LIN {X 0,Y 401.076,Z 526.774,A -85,B 0,C 180,E1 -11232.866,E2 -11232.866} C_VEL
LIN {X 0,Y 400.137,Z 539.303,A -85,B 0,C 180,E1 -11233.547,E2 -11233.547} C_VEL
LIN {X 0,Y 399.29,Z 551.619,A -85,B 0,C 180,E1 -11234.43,E2 -11234.43} C_VEL
LIN {X 0,Y 398.339,Z 562.751,A -85,B 0,C 180,E1 -11235.438,E2 -11235.438} C_VEL
LIN {X 0,Y 397.548,Z 573.979,A -85,B 0,C 180,E1 -11236.713,E2 -11236.713} C_VEL
LIN {X 0,Y 397.078,Z 581.427,A -85,B 0,C 180,E1 -11237.737,E2 -11237.737} C_VEL
LIN {X 0,Y 396.635,Z 590.764,A -85,B 0,C 180,E1 -11239.277,E2 -11239.277} C_VEL
LIN {X 0,Y 396.29,Z 600.831,A -85,B 0,C 180,E1 -11241.33,E2 -11241.33} C_VEL
LIN {X 0,Y 396.234,Z 606.786,A -85,B 0,C 180,E1 -11242.868,E2 -11242.868} C_VEL
LIN {X 0,Y 396.252,Z 611.402,A -85,B 0,C 180,E1 -11244.402,E2 -11244.402} C_VEL
LIN {X 0,Y 396.439,Z 614.849,A -85,B 0,C 180,E1 -11245.933,E2 -11245.933} C_VEL
LIN {X 0,Y 396.415,Z 616.498,A -85,B 0,C 180,E1 -11246.951,E2 -11246.951} C_VEL
LIN {X 0,Y 396.382,Z 617.7,A -85,B 0,C 180,E1 -11247.968,E2 -11247.968} C_VEL
LIN {X 0,Y 396.396,Z 618.449,A -85,B 0,C 180,E1 -11248.984,E2 -11248.984} C_VEL
LIN {X 0,Y 396.436,Z 618.72,A -85,B 0,C 180,E1 -11250,E2 -11250} C_VEL
LIN {X 0,Y 396.383,Z 618.544,A -85,B 0,C 180,E1 -11251.016,E2 -11251.016} C_VEL
LIN {X 0,Y 396.351,Z 617.942,A -85,B 0,C 180,E1 -11252.032,E2 -11252.032} C_VEL
LIN {X 0,Y 396.408,Z 616.87,A -85,B 0,C 180,E1 -11253.049,E2 -11253.049} C_VEL
LIN {X 0,Y 396.385,Z 615.337,A -85,B 0,C 180,E1 -11254.067,E2 -11254.067} C_VEL
LIN {X 0,Y 396.242,Z 612.157,A -85,B 0,C 180,E1 -11255.598,E2 -11255.598} C_VEL
LIN {X 0,Y 396.214,Z 607.863,A -85,B 0,C 180,E1 -11257.132,E2 -11257.132} C_VEL
LIN {X 0,Y 396.243,Z 602.363,A -85,B 0,C 180,E1 -11258.671,E2 -11258.671} C_VEL
LIN {X 0,Y 396.426,Z 595.508,A -85,B 0,C 180,E1 -11260.211,E2 -11260.211} C_VEL
LIN {X 0,Y 396.908,Z 587.032,A -85,B 0,C 180,E1 -11261.749,E2 -11261.749} C_VEL
LIN {X 0,Y 397.568,Z 578.464,A -85,B 0,C 180,E1 -11263.026,E2 -11263.026} C_VEL
LIN {X 0,Y 398.292,Z 568.093,A -85,B 0,C 180,E1 -11264.302,E2 -11264.302} C_VEL
LIN {X 0,Y 399.23,Z 556.682,A -85,B 0,C 180,E1 -11265.442,E2 -11265.442} C_VEL
LIN {X 0,Y 400.376,Z 543.918,A -85,B 0,C 180,E1 -11266.442,E2 -11266.442} C_VEL
LIN {X 0,Y 401.252,Z 531.695,A -85,B 0,C 180,E1 -11267.192,E2 -11267.192} C_VEL
LIN {X 0,Y 402.229,Z 517.827,A -85,B 0,C 180,E1 -11267.804,E2 -11267.804} C_VEL
LIN {X 0,Y 402.722,Z 503.308,A -85,B 0,C 180,E1 -11268.242,E2 -11268.242} C_VEL
LIN {X 0,Y 404.434,Z 442.131,A -85,B 0,C 180,E1 -11269.695,E2 -11269.695} C_VEL
LIN {X 0,Y 402.5,Z 418.971,A -85,B 0,C 180,E1 -11270.461,E2 -11270.461} C_VEL
LIN {X 0,Y 400.143,Z 402.554,A -85,B 0,C 180,E1 -11271.103,E2 -11271.103} C_VEL
LIN {X 0,Y 399.183,Z 396.5,A -85,B 0,C 180,E1 -11271.372,E2 -11271.372} C_VEL
LIN {X 0,Y 400.84,Z 376.396,A -85,B 0,C 180,E1 -11274.885,E2 -11274.885} C_VEL
LIN {X 0,Y 402.863,Z 357.39,A -85,B 0,C 180,E1 -11278.362,E2 -11278.362} C_VEL
LIN {X 0,Y 402.396,Z 353.06,A -85,B 0,C 180,E1 -11279.277,E2 -11279.277} C_VEL
LIN {X 0,Y 400.617,Z 344.823,A -85,B 0,C 180,E1 -11281.177,E2 -11281.177} C_VEL
LIN {X 0,Y 398.111,Z 335.577,A -85,B 0,C 180,E1 -11283.57,E2 -11283.57} C_VEL
LIN {X 0,Y 397.129,Z 332.018,A -85,B 0,C 180,E1 -11284.608,E2 -11284.608} C_VEL
LIN {X 0,Y 397.094,Z 332.024,A -85,B 0,C 180,E1 -11288.276,E2 -11288.276} C_VEL
LIN {X 0,Y 397.056,Z 332.029,A -85,B 0,C 180,E1 -11291.977,E2 -11291.977} C_VEL
LIN {X 0,Y 397.088,Z 332.023,A -85,B 0,C 180,E1 -11295.069,E2 -11295.069} C_VEL
LIN {X 0,Y 397.055,Z 332.028,A -85,B 0,C 180,E1 -11298.023,E2 -11298.023} C_VEL
LIN {X 0,Y 397.091,Z 332.022,A -85,B 0,C 180,E1 -11301.723,E2 -11301.723} C_VEL
LIN {X 0,Y 397.118,Z 332.018,A -85,B 0,C 180,E1 -11305.506,E2 -11305.506} C_VEL
LIN {X 0,Y 397.078,Z 332.024,A -85,B 0,C 180,E1 -11309.117,E2 -11309.117} C_VEL
LIN {X 0,Y 397.061,Z 332.027,A -85,B 0,C 180,E1 -11312.252,E2 -11312.252} C_VEL
LIN {X 0,Y 397.103,Z 332.022,A -85,B 0,C 180,E1 -11314.864,E2 -11314.864} C_VEL
LIN {X 0,Y 397.091,Z 332.026,A -85,B 0,C 180,E1 -11318.181,E2 -11318.181} C_VEL
LIN {X 0,Y 397.127,Z 332.217,A -85,B 0,C 180,E1 -11320.855,E2 -11320.855} C_VEL
LIN {X 0,Y 398.352,Z 335.23,A -85,B 0,C 180,E1 -11321.058,E2 -11321.058} C_VEL
LIN {X 0,Y 404.412,Z 347.267,A -85,B 0,C 180,E1 -11321.939,E2 -11321.939} C_VEL
LIN {X 0,Y 406.246,Z 351.624,A -85,B 0,C 180,E1 -11322.213,E2 -11322.213} C_VEL
LIN {X 0,Y 404.005,Z 419.893,A -85,B 0,C 180,E1 -11323.904,E2 -11323.904} C_VEL
LIN {X 0,Y 403.82,Z 433.902,A -85,B 0,C 180,E1 -11324.382,E2 -11324.382} C_VEL
LIN {X 0,Y 403.426,Z 446.94,A -85,B 0,C 180,E1 -11325.045,E2 -11325.045} C_VEL
LIN {X 0,Y 402.874,Z 458.91,A -85,B 0,C 180,E1 -11325.863,E2 -11325.863} C_VEL
LIN {X 0,Y 402.114,Z 470.396,A -85,B 0,C 180,E1 -11326.867,E2 -11326.867} C_VEL
LIN {X 0,Y 401.281,Z 481.639,A -85,B 0,C 180,E1 -11328.124,E2 -11328.124} C_VEL
LIN {X 0,Y 400.417,Z 491.372,A -85,B 0,C 180,E1 -11329.483,E2 -11329.483} C_VEL
LIN {X 0,Y 399.587,Z 499.48,A -85,B 0,C 180,E1 -11330.892,E2 -11330.892} C_VEL
LIN {X 0,Y 398.939,Z 506.463,A -85,B 0,C 180,E1 -11332.407,E2 -11332.407} C_VEL
LIN {X 0,Y 398.197,Z 512.05,A -85,B 0,C 180,E1 -11333.921,E2 -11333.921} C_VEL
LIN {X 0,Y 397.8,Z 516.329,A -85,B 0,C 180,E1 -11335.44,E2 -11335.44} C_VEL
LIN {X 0,Y 397.367,Z 519.526,A -85,B 0,C 180,E1 -11336.958,E2 -11336.958} C_VEL
LIN {X 0,Y 397.258,Z 521.043,A -85,B 0,C 180,E1 -11337.972,E2 -11337.972} C_VEL
LIN {X 0,Y 397.11,Z 522.162,A -85,B 0,C 180,E1 -11338.985,E2 -11338.985} C_VEL
LIN {X 0,Y 396.984,Z 522.869,A -85,B 0,C 180,E1 -11340,E2 -11340} C_VEL
LIN {X 0,Y 396.873,Z 523.115,A -85,B 0,C 180,E1 -11341.014,E2 -11341.014} C_VEL
LIN {X 0,Y 396.586,Z 522.978,A -85,B 0,C 180,E1 -11342.031,E2 -11342.031} C_VEL
LIN {X 0,Y 396.606,Z 522.4,A -85,B 0,C 180,E1 -11343.047,E2 -11343.047} C_VEL
LIN {X 0,Y 396.737,Z 521.37,A -85,B 0,C 180,E1 -11344.063,E2 -11344.063} C_VEL
LIN {X 0,Y 396.891,Z 519.903,A -85,B 0,C 180,E1 -11345.079,E2 -11345.079} C_VEL
LIN {X 0,Y 396.972,Z 516.904,A -85,B 0,C 180,E1 -11346.608,E2 -11346.608} C_VEL
LIN {X 0,Y 397.143,Z 512.82,A -85,B 0,C 180,E1 -11348.138,E2 -11348.138} C_VEL
LIN {X 0,Y 397.411,Z 507.538,A -85,B 0,C 180,E1 -11349.671,E2 -11349.671} C_VEL
LIN {X 0,Y 397.757,Z 500.899,A -85,B 0,C 180,E1 -11351.207,E2 -11351.207} C_VEL
LIN {X 0,Y 398.266,Z 492.555,A -85,B 0,C 180,E1 -11352.743,E2 -11352.743} C_VEL
LIN {X 0,Y 398.681,Z 484.171,A -85,B 0,C 180,E1 -11354.007,E2 -11354.007} C_VEL
LIN {X 0,Y 399.248,Z 473.607,A -85,B 0,C 180,E1 -11355.31,E2 -11355.31} C_VEL
LIN {X 0,Y 399.815,Z 461.79,A -85,B 0,C 180,E1 -11356.466,E2 -11356.466} C_VEL
LIN {X 0,Y 400.32,Z 450.233,A -85,B 0,C 180,E1 -11357.364,E2 -11357.364} C_VEL
LIN {X 0,Y 400.771,Z 437.173,A -85,B 0,C 180,E1 -11358.135,E2 -11358.135} C_VEL
LIN {X 0,Y 400.998,Z 423.42,A -85,B 0,C 180,E1 -11358.721,E2 -11358.721} C_VEL
LIN {X 0,Y 401.168,Z 408.327,A -85,B 0,C 180,E1 -11359.115,E2 -11359.115} C_VEL
LIN {X 0,Y 402.218,Z 347.343,A -85,B 0,C 180,E1 -11360.446,E2 -11360.446} C_VEL
LIN {X 0,Y 397.121,Z 332.019,A -85,B 0,C 180,E1 -11361.015,E2 -11361.015} C_VEL
LIN {X 0,Y 397.133,Z 332.014,A -85,B 0,C 180,E1 -11364.018,E2 -11364.018} C_VEL
LIN {X 0,Y 397.194,Z 332.007,A -85,B 0,C 180,E1 -11367.39,E2 -11367.39} C_VEL
LIN {X 0,Y 397.078,Z 332.025,A -85,B 0,C 180,E1 -11370.882,E2 -11370.882} C_VEL
LIN {X 0,Y 397.124,Z 332.018,A -85,B 0,C 180,E1 -11374.493,E2 -11374.493} C_VEL
LIN {X 0,Y 397.099,Z 332.02,A -85,B 0,C 180,E1 -11378.275,E2 -11378.275} C_VEL
LIN {X 0,Y 397.087,Z 332.023,A -85,B 0,C 180,E1 -11380.908,E2 -11380.908} C_VEL
LIN {X 0,Y 397.099,Z 332.018,A -85,B 0,C 180,E1 -11383.648,E2 -11383.648} C_VEL
LIN {X 0,Y 397.1,Z 332.022,A -85,B 0,C 180,E1 -11386.521,E2 -11386.521} C_VEL
LIN {X 0,Y 397.113,Z 332.02,A -85,B 0,C 180,E1 -11390.423,E2 -11390.423} C_VEL
LIN {X 0,Y 397.107,Z 332.02,A -85,B 0,C 180,E1 -11394.265,E2 -11394.265} C_VEL
LIN {X 0,Y 397.112,Z 332.02,A -85,B 0,C 180,E1 -11396.727,E2 -11396.727} C_VEL
LIN {X 0,Y 397.122,Z 332.019,A -85,B 0,C 180,E1 -11400.296,E2 -11400.296} C_VEL
LIN {X 0,Y 397.192,Z 332.011,A -85,B 0,C 180,E1 -11402.61,E2 -11402.61} C_VEL
LIN {X 0,Y 397.13,Z 332.015,A -85,B 0,C 180,E1 -11405.982,E2 -11405.982} C_VEL
LIN {X 0,Y 397.136,Z 332.014,A -85,B 0,C 180,E1 -11409.704,E2 -11409.704} C_VEL
LIN {X 0,Y 397.179,Z 332.01,A -85,B 0,C 180,E1 -11412.845,E2 -11412.845} C_VEL
LIN {X 0,Y 397.226,Z 332.005,A -85,B 0,C 180,E1 -11416.703,E2 -11416.703} C_VEL
LIN {X 0,Y 397.221,Z 332.004,A -85,B 0,C 180,E1 -11419.809,E2 -11419.809} C_VEL
LIN {X 0,Y 397.361,Z 331.987,A -85,B 0,C 180,E1 -11422.888,E2 -11422.888} C_VEL
LIN {X 0,Y 397.252,Z 332,A -85,B 0,C 180,E1 -11424.925,E2 -11424.925} C_VEL
LIN {X 0,Y 397.449,Z 331.977,A -85,B 0,C 180,E1 -11427.973,E2 -11427.973} C_VEL
LIN {X 0,Y 397.578,Z 331.961,A -85,B 0,C 180,E1 -11430,E2 -11430} C_VEL
LIN {X 0,Y 397.379,Z 331.984,A -85,B 0,C 180,E1 -11433.042,E2 -11433.042} C_VEL
LIN {X 0,Y 397.362,Z 331.986,A -85,B 0,C 180,E1 -11437.112,E2 -11437.112} C_VEL
LIN {X 0,Y 397.216,Z 332.009,A -85,B 0,C 180,E1 -11440.191,E2 -11440.191} C_VEL
LIN {X 0,Y 397.224,Z 332.003,A -85,B 0,C 180,E1 -11443.321,E2 -11443.321} C_VEL
LIN {X 0,Y 397.166,Z 332.012,A -85,B 0,C 180,E1 -11444.49,E2 -11444.49} C_VEL
LIN {X 0,Y 396.488,Z 332.095,A -85,B 0,C 180,E1 -11445.337,E2 -11445.337} C_VEL
LIN {X 0,Y 393.652,Z 332.449,A -85,B 0,C 180,E1 -11446.714,E2 -11446.714} C_VEL
LIN {X 0,Y 391.247,Z 332.75,A -85,B 0,C 180,E1 -11447.826,E2 -11447.826} C_VEL
LIN {X 0,Y 390.196,Z 332.88,A -85,B 0,C 180,E1 -11448.686,E2 -11448.686} C_VEL
LIN {X 0,Y 390.1,Z 332.891,A -85,B 0,C 180,E1 -11448.977,E2 -11448.977} C_VEL
LIN {X 0,Y 390.039,Z 332.902,A -85,B 0,C 180,E1 -11452.235,E2 -11452.235} C_VEL
LIN {X 0,Y 390.118,Z 332.89,A -85,B 0,C 180,E1 -11455.744,E2 -11455.744} C_VEL
LIN {X 0,Y 390.057,Z 332.896,A -85,B 0,C 180,E1 -11459.11,E2 -11459.11} C_VEL
LIN {X 0,Y 390.042,Z 332.899,A -85,B 0,C 180,E1 -11462.722,E2 -11462.722} C_VEL
LIN {X 0,Y 390.057,Z 332.899,A -85,B 0,C 180,E1 -11465.826,E2 -11465.826} C_VEL
LIN {X 0,Y 390.071,Z 332.894,A -85,B 0,C 180,E1 -11469.219,E2 -11469.219} C_VEL
LIN {X 0,Y 390.042,Z 332.899,A -85,B 0,C 180,E1 -11472.375,E2 -11472.375} C_VEL
LIN {X 0,Y 390.044,Z 332.898,A -85,B 0,C 180,E1 -11475.355,E2 -11475.355} C_VEL
LIN {X 0,Y 390.031,Z 332.901,A -85,B 0,C 180,E1 -11478.187,E2 -11478.187} C_VEL
LIN {X 0,Y 390.088,Z 332.892,A -85,B 0,C 180,E1 -11480.908,E2 -11480.908} C_VEL
LIN {X 0,Y 390.085,Z 332.892,A -85,B 0,C 180,E1 -11484.794,E2 -11484.794} C_VEL
LIN {X 0,Y 390.025,Z 332.901,A -85,B 0,C 180,E1 -11488.496,E2 -11488.496} C_VEL
LIN {X 0,Y 390.141,Z 332.887,A -85,B 0,C 180,E1 -11492.454,E2 -11492.454} C_VEL
LIN {X 0,Y 390.171,Z 332.883,A -85,B 0,C 180,E1 -11492.773,E2 -11492.773} C_VEL
LIN {X 0,Y 395.504,Z 349.657,A -85,B 0,C 180,E1 -11493.387,E2 -11493.387} C_VEL
LIN {X 0,Y 394.229,Z 420.499,A -85,B 0,C 180,E1 -11494.955,E2 -11494.955} C_VEL
LIN {X 0,Y 394.109,Z 433.109,A -85,B 0,C 180,E1 -11495.433,E2 -11495.433} C_VEL
LIN {X 0,Y 393.68,Z 446.836,A -85,B 0,C 180,E1 -11496.178,E2 -11496.178} C_VEL
LIN {X 0,Y 393.245,Z 458.09,A -85,B 0,C 180,E1 -11496.987,E2 -11496.987} C_VEL
LIN {X 0,Y 392.653,Z 469.556,A -85,B 0,C 180,E1 -11498.036,E2 -11498.036} C_VEL
LIN {X 0,Y 392.075,Z 480.383,A -85,B 0,C 180,E1 -11499.267,E2 -11499.267} C_VEL
LIN {X 0,Y 391.417,Z 489.829,A -85,B 0,C 180,E1 -11500.6,E2 -11500.6} C_VEL
LIN {X 0,Y 390.898,Z 499.025,A -85,B 0,C 180,E1 -11502.204,E2 -11502.204} C_VEL
LIN {X 0,Y 390.473,Z 506.266,A -85,B 0,C 180,E1 -11503.801,E2 -11503.801} C_VEL
LIN {X 0,Y 390.11,Z 512.029,A -85,B 0,C 180,E1 -11505.392,E2 -11505.392} C_VEL
LIN {X 0,Y 389.964,Z 515.798,A -85,B 0,C 180,E1 -11506.707,E2 -11506.707} C_VEL
LIN {X 0,Y 389.705,Z 519.817,A -85,B 0,C 180,E1 -11508.559,E2 -11508.559} C_VEL
LIN {X 0,Y 389.664,Z 521.416,A -85,B 0,C 180,E1 -11509.61,E2 -11509.61} C_VEL
LIN {X 0,Y 389.685,Z 522.576,A -85,B 0,C 180,E1 -11510.659,E2 -11510.659} C_VEL
LIN {X 0,Y 389.818,Z 523.599,A -85,B 0,C 180,E1 -11512.569,E2 -11512.569} C_VEL
LIN {X 0,Y 389.885,Z 523.466,A -85,B 0,C 180,E1 -11513.792,E2 -11513.792} C_VEL
LIN {X 0,Y 389.936,Z 522.938,A -85,B 0,C 180,E1 -11514.83,E2 -11514.83} C_VEL
LIN {X 0,Y 390.019,Z 521.955,A -85,B 0,C 180,E1 -11515.867,E2 -11515.867} C_VEL
LIN {X 0,Y 390.272,Z 520.52,A -85,B 0,C 180,E1 -11516.904,E2 -11516.904} C_VEL
LIN {X 0,Y 390.686,Z 517.544,A -85,B 0,C 180,E1 -11518.454,E2 -11518.454} C_VEL
LIN {X 0,Y 391.202,Z 513.483,A -85,B 0,C 180,E1 -11520,E2 -11520} C_VEL
LIN {X 0,Y 391.814,Z 508.228,A -85,B 0,C 180,E1 -11521.542,E2 -11521.542} C_VEL
LIN {X 0,Y 392.496,Z 501.585,A -85,B 0,C 180,E1 -11523.08,E2 -11523.08} C_VEL
LIN {X 0,Y 393.4,Z 493.235,A -85,B 0,C 180,E1 -11524.612,E2 -11524.612} C_VEL
LIN {X 0,Y 394.145,Z 484.749,A -85,B 0,C 180,E1 -11525.885,E2 -11525.885} C_VEL
LIN {X 0,Y 395.074,Z 474.19,A -85,B 0,C 180,E1 -11527.154,E2 -11527.154} C_VEL
LIN {X 0,Y 395.801,Z 463.747,A -85,B 0,C 180,E1 -11528.167,E2 -11528.167} C_VEL
LIN {X 0,Y 396.475,Z 452.162,A -85,B 0,C 180,E1 -11529.052,E2 -11529.052} C_VEL
LIN {X 0,Y 396.942,Z 439.066,A -85,B 0,C 180,E1 -11529.812,E2 -11529.812} C_VEL
LIN {X 0,Y 397.177,Z 426.656,A -85,B 0,C 180,E1 -11530.321,E2 -11530.321} C_VEL
LIN {X 0,Y 397.828,Z 396.469,A -85,B 0,C 180,E1 -11531.077,E2 -11531.077} C_VEL
LIN {X 0,Y 399.244,Z 352.593,A -85,B 0,C 180,E1 -11532.149,E2 -11532.149} C_VEL
LIN {X 0,Y 392.78,Z 338.726,A -85,B 0,C 180,E1 -11533.068,E2 -11533.068} C_VEL
LIN {X 0,Y 390.316,Z 333.585,A -85,B 0,C 180,E1 -11533.44,E2 -11533.44} C_VEL
LIN {X 0,Y 390.172,Z 332.884,A -85,B 0,C 180,E1 -11533.483,E2 -11533.483} C_VEL
LIN {X 0,Y 390.131,Z 332.89,A -85,B 0,C 180,E1 -11536.753,E2 -11536.753} C_VEL
LIN {X 0,Y 390.071,Z 332.898,A -85,B 0,C 180,E1 -11540.462,E2 -11540.462} C_VEL
LIN {X 0,Y 390.06,Z 332.896,A -85,B 0,C 180,E1 -11543.353,E2 -11543.353} C_VEL
LIN {X 0,Y 390.031,Z 332.903,A -85,B 0,C 180,E1 -11546.775,E2 -11546.775} C_VEL
LIN {X 0,Y 390.04,Z 332.901,A -85,B 0,C 180,E1 -11550.3,E2 -11550.3} C_VEL
LIN {X 0,Y 390.073,Z 332.896,A -85,B 0,C 180,E1 -11554.025,E2 -11554.025} C_VEL
LIN {X 0,Y 390.039,Z 332.898,A -85,B 0,C 180,E1 -11557.781,E2 -11557.781} C_VEL
LIN {X 0,Y 390.02,Z 332.897,A -85,B 0,C 180,E1 -11560.814,E2 -11560.814} C_VEL
LIN {X 0,Y 390.047,Z 332.898,A -85,B 0,C 180,E1 -11563.884,E2 -11563.884} C_VEL
LIN {X 0,Y 390.056,Z 332.897,A -85,B 0,C 180,E1 -11566.789,E2 -11566.789} C_VEL
LIN {X 0,Y 390.013,Z 332.906,A -85,B 0,C 180,E1 -11569.555,E2 -11569.555} C_VEL
LIN {X 0,Y 390.043,Z 332.899,A -85,B 0,C 180,E1 -11572.45,E2 -11572.45} C_VEL
LIN {X 0,Y 390.072,Z 332.898,A -85,B 0,C 180,E1 -11575.975,E2 -11575.975} C_VEL
LIN {X 0,Y 390.082,Z 332.9,A -85,B 0,C 180,E1 -11577.528,E2 -11577.528} C_VEL
LIN {X 0,Y 393.929,Z 350.251,A -85,B 0,C 180,E1 -11580.81,E2 -11580.81} C_VEL
LIN {X 0,Y 394.861,Z 356.022,A -85,B 0,C 180,E1 -11581.857,E2 -11581.857} C_VEL
LIN {X 0,Y 393.22,Z 377.335,A -85,B 0,C 180,E1 -11585.446,E2 -11585.446} C_VEL
LIN {X 0,Y 391.915,Z 396.452,A -85,B 0,C 180,E1 -11588.636,E2 -11588.636} C_VEL
LIN {X 0,Y 395.233,Z 422.029,A -85,B 0,C 180,E1 -11589.597,E2 -11589.597} C_VEL
LIN {X 0,Y 397.032,Z 444.166,A -85,B 0,C 180,E1 -11590.313,E2 -11590.313} C_VEL
LIN {X 0,Y 395.175,Z 511.505,A -85,B 0,C 180,E1 -11591.933,E2 -11591.933} C_VEL
LIN {X 0,Y 394.488,Z 524.712,A -85,B 0,C 180,E1 -11592.437,E2 -11592.437} C_VEL
LIN {X 0,Y 393.515,Z 537.528,A -85,B 0,C 180,E1 -11593.129,E2 -11593.129} C_VEL
LIN {X 0,Y 392.552,Z 549.936,A -85,B 0,C 180,E1 -11594.022,E2 -11594.022} C_VEL
LIN {X 0,Y 391.551,Z 561.181,A -85,B 0,C 180,E1 -11595.047,E2 -11595.047} C_VEL
LIN {X 0,Y 390.72,Z 571.689,A -85,B 0,C 180,E1 -11596.245,E2 -11596.245} C_VEL
LIN {X 0,Y 390.116,Z 580.882,A -85,B 0,C 180,E1 -11597.515,E2 -11597.515} C_VEL
LIN {X 0,Y 389.672,Z 588.72,A -85,B 0,C 180,E1 -11598.82,E2 -11598.82} C_VEL
LIN {X 0,Y 389.31,Z 596.446,A -85,B 0,C 180,E1 -11600.387,E2 -11600.387} C_VEL
LIN {X 0,Y 389.191,Z 605.603,A -85,B 0,C 180,E1 -11602.738,E2 -11602.738} C_VEL
LIN {X 0,Y 389.203,Z 610.301,A -85,B 0,C 180,E1 -11604.3,E2 -11604.3} C_VEL
LIN {X 0,Y 389.369,Z 613.81,A -85,B 0,C 180,E1 -11605.86,E2 -11605.86} C_VEL
LIN {X 0,Y 389.371,Z 615.489,A -85,B 0,C 180,E1 -11606.896,E2 -11606.896} C_VEL
LIN {X 0,Y 389.342,Z 616.717,A -85,B 0,C 180,E1 -11607.931,E2 -11607.931} C_VEL
LIN {X 0,Y 389.355,Z 617.506,A -85,B 0,C 180,E1 -11608.966,E2 -11608.966} C_VEL
LIN {X 0,Y 389.394,Z 617.807,A -85,B 0,C 180,E1 -11610,E2 -11610} C_VEL
LIN {X 0,Y 389.335,Z 617.651,A -85,B 0,C 180,E1 -11611.034,E2 -11611.034} C_VEL
LIN {X 0,Y 389.3,Z 617.065,A -85,B 0,C 180,E1 -11612.069,E2 -11612.069} C_VEL
LIN {X 0,Y 389.362,Z 616.036,A -85,B 0,C 180,E1 -11613.104,E2 -11613.104} C_VEL
LIN {X 0,Y 389.315,Z 614.512,A -85,B 0,C 180,E1 -11614.141,E2 -11614.141} C_VEL
LIN {X 0,Y 389.177,Z 611.37,A -85,B 0,C 180,E1 -11615.7,E2 -11615.7} C_VEL
LIN {X 0,Y 389.122,Z 607.117,A -85,B 0,C 180,E1 -11617.263,E2 -11617.263} C_VEL
LIN {X 0,Y 389.184,Z 600.632,A -85,B 0,C 180,E1 -11619.091,E2 -11619.091} C_VEL
LIN {X 0,Y 389.467,Z 593.595,A -85,B 0,C 180,E1 -11620.659,E2 -11620.659} C_VEL
LIN {X 0,Y 389.975,Z 584.867,A -85,B 0,C 180,E1 -11622.225,E2 -11622.225} C_VEL
LIN {X 0,Y 390.675,Z 576.087,A -85,B 0,C 180,E1 -11623.524,E2 -11623.524} C_VEL
LIN {X 0,Y 391.529,Z 565.471,A -85,B 0,C 180,E1 -11624.82,E2 -11624.82} C_VEL
LIN {X 0,Y 392.644,Z 553.632,A -85,B 0,C 180,E1 -11625.974,E2 -11625.974} C_VEL
LIN {X 0,Y 393.715,Z 542.263,A -85,B 0,C 180,E1 -11626.862,E2 -11626.862} C_VEL
LIN {X 0,Y 394.719,Z 529.925,A -85,B 0,C 180,E1 -11627.619,E2 -11627.619} C_VEL
LIN {X 0,Y 395.757,Z 515.074,A -85,B 0,C 180,E1 -11628.273,E2 -11628.273} C_VEL
LIN {X 0,Y 396.287,Z 499.824,A -85,B 0,C 180,E1 -11628.716,E2 -11628.716} C_VEL
LIN {X 0,Y 398.005,Z 442.029,A -85,B 0,C 180,E1 -11630.142,E2 -11630.142} C_VEL
LIN {X 0,Y 396.121,Z 419.552,A -85,B 0,C 180,E1 -11630.922,E2 -11630.922} C_VEL
LIN {X 0,Y 393.92,Z 403.885,A -85,B 0,C 180,E1 -11631.561,E2 -11631.561} C_VEL
LIN {X 0,Y 392.425,Z 395.103,A -85,B 0,C 180,E1 -11631.974,E2 -11631.974} C_VEL
LIN {X 0,Y 394.121,Z 376.402,A -85,B 0,C 180,E1 -11635.339,E2 -11635.339} C_VEL
LIN {X 0,Y 396.167,Z 358.967,A -85,B 0,C 180,E1 -11638.619,E2 -11638.619} C_VEL
LIN {X 0,Y 395.385,Z 353.418,A -85,B 0,C 180,E1 -11639.848,E2 -11639.848} C_VEL
LIN {X 0,Y 393.264,Z 344.177,A -85,B 0,C 180,E1 -11642.117,E2 -11642.117} C_VEL
LIN {X 0,Y 390.833,Z 335.431,A -85,B 0,C 180,E1 -11644.559,E2 -11644.559} C_VEL
LIN {X 0,Y 390.111,Z 332.894,A -85,B 0,C 180,E1 -11645.358,E2 -11645.358} C_VEL
LIN {X 0,Y 390.039,Z 332.903,A -85,B 0,C 180,E1 -11649.212,E2 -11649.212} C_VEL
LIN {X 0,Y 390.034,Z 332.903,A -85,B 0,C 180,E1 -11652.372,E2 -11652.372} C_VEL
LIN {X 0,Y 390.045,Z 332.9,A -85,B 0,C 180,E1 -11655.354,E2 -11655.354} C_VEL
LIN {X 0,Y 390.018,Z 332.904,A -85,B 0,C 180,E1 -11658.184,E2 -11658.184} C_VEL
LIN {X 0,Y 390.058,Z 332.896,A -85,B 0,C 180,E1 -11660.903,E2 -11660.903} C_VEL
LIN {X 0,Y 390.07,Z 332.895,A -85,B 0,C 180,E1 -11664.791,E2 -11664.791} C_VEL
LIN {X 0,Y 390.023,Z 332.903,A -85,B 0,C 180,E1 -11668.495,E2 -11668.495} C_VEL
LIN {X 0,Y 390.017,Z 332.906,A -85,B 0,C 180,E1 -11672.003,E2 -11672.003} C_VEL
LIN {X 0,Y 390.043,Z 332.904,A -85,B 0,C 180,E1 -11675.516,E2 -11675.516} C_VEL
LIN {X 0,Y 390.051,Z 332.901,A -85,B 0,C 180,E1 -11678.877,E2 -11678.877} C_VEL
LIN {X 0,Y 390.067,Z 332.897,A -85,B 0,C 180,E1 -11680.198,E2 -11680.198} C_VEL
LIN {X 0,Y 391.11,Z 335.827,A -85,B 0,C 180,E1 -11680.4,E2 -11680.4} C_VEL
LIN {X 0,Y 395.384,Z 343.748,A -85,B 0,C 180,E1 -11681.058,E2 -11681.058} C_VEL
LIN {X 0,Y 400.014,Z 353.673,A -85,B 0,C 180,E1 -11681.766,E2 -11681.766} C_VEL
LIN {X 0,Y 397.59,Z 419.705,A -85,B 0,C 180,E1 -11683.455,E2 -11683.455} C_VEL
LIN {X 0,Y 397.429,Z 433.64,A -85,B 0,C 180,E1 -11683.927,E2 -11683.927} C_VEL
LIN {X 0,Y 397.067,Z 445.914,A -85,B 0,C 180,E1 -11684.537,E2 -11684.537} C_VEL
LIN {X 0,Y 396.429,Z 458.357,A -85,B 0,C 180,E1 -11685.366,E2 -11685.366} C_VEL
LIN {X 0,Y 395.657,Z 470.132,A -85,B 0,C 180,E1 -11686.387,E2 -11686.387} C_VEL
LIN {X 0,Y 394.825,Z 480.61,A -85,B 0,C 180,E1 -11687.535,E2 -11687.535} C_VEL
LIN {X 0,Y 393.958,Z 490.371,A -85,B 0,C 180,E1 -11688.865,E2 -11688.865} C_VEL
LIN {X 0,Y 393.076,Z 498.783,A -85,B 0,C 180,E1 -11690.277,E2 -11690.277} C_VEL
LIN {X 0,Y 392.201,Z 505.868,A -85,B 0,C 180,E1 -11691.757,E2 -11691.757} C_VEL
LIN {X 0,Y 391.557,Z 511.729,A -85,B 0,C 180,E1 -11693.3,E2 -11693.3} C_VEL
LIN {X 0,Y 390.961,Z 516.326,A -85,B 0,C 180,E1 -11694.843,E2 -11694.843} C_VEL
LIN {X 0,Y 390.656,Z 518.768,A -85,B 0,C 180,E1 -11695.873,E2 -11695.873} C_VEL
LIN {X 0,Y 390.382,Z 520.701,A -85,B 0,C 180,E1 -11696.904,E2 -11696.904} C_VEL
LIN {X 0,Y 390.253,Z 522.172,A -85,B 0,C 180,E1 -11697.935,E2 -11697.935} C_VEL
LIN {X 0,Y 390.098,Z 523.24,A -85,B 0,C 180,E1 -11698.967,E2 -11698.967} C_VEL
LIN {X 0,Y 389.975,Z 523.861,A -85,B 0,C 180,E1 -11700,E2 -11700} C_VEL
LIN {X 0,Y 389.839,Z 524.052,A -85,B 0,C 180,E1 -11701.032,E2 -11701.032} C_VEL
LIN {X 0,Y 389.543,Z 523.864,A -85,B 0,C 180,E1 -11702.067,E2 -11702.067} C_VEL
LIN {X 0,Y 389.562,Z 523.222,A -85,B 0,C 180,E1 -11703.102,E2 -11703.102} C_VEL
LIN {X 0,Y 389.708,Z 522.109,A -85,B 0,C 180,E1 -11704.136,E2 -11704.136} C_VEL
LIN {X 0,Y 389.847,Z 520.588,A -85,B 0,C 180,E1 -11705.171,E2 -11705.171} C_VEL
LIN {X 0,Y 389.917,Z 517.481,A -85,B 0,C 180,E1 -11706.728,E2 -11706.728} C_VEL
LIN {X 0,Y 390.125,Z 513.277,A -85,B 0,C 180,E1 -11708.286,E2 -11708.286} C_VEL
LIN {X 0,Y 390.389,Z 507.867,A -85,B 0,C 180,E1 -11709.847,E2 -11709.847} C_VEL
LIN {X 0,Y 390.776,Z 501.038,A -85,B 0,C 180,E1 -11711.41,E2 -11711.41} C_VEL
LIN {X 0,Y 391.305,Z 492.513,A -85,B 0,C 180,E1 -11712.973,E2 -11712.973} C_VEL
LIN {X 0,Y 391.805,Z 482.992,A -85,B 0,C 180,E1 -11714.39,E2 -11714.39} C_VEL
LIN {X 0,Y 392.327,Z 471.819,A -85,B 0,C 180,E1 -11715.72,E2 -11715.72} C_VEL
LIN {X 0,Y 392.912,Z 460.92,A -85,B 0,C 180,E1 -11716.763,E2 -11716.763} C_VEL
LIN {X 0,Y 393.46,Z 448.796,A -85,B 0,C 180,E1 -11717.677,E2 -11717.677} C_VEL
LIN {X 0,Y 393.88,Z 436.35,A -85,B 0,C 180,E1 -11718.396,E2 -11718.396} C_VEL
LIN {X 0,Y 394.07,Z 423.252,A -85,B 0,C 180,E1 -11718.943,E2 -11718.943} C_VEL
LIN {X 0,Y 394.278,Z 406.24,A -85,B 0,C 180,E1 -11719.377,E2 -11719.377} C_VEL
LIN {X 0,Y 395.265,Z 348.568,A -85,B 0,C 180,E1 -11720.67,E2 -11720.67} C_VEL
LIN {X 0,Y 390.077,Z 332.895,A -85,B 0,C 180,E1 -11721.257,E2 -11721.257} C_VEL
LIN {X 0,Y 390.081,Z 332.894,A -85,B 0,C 180,E1 -11724.48,E2 -11724.48} C_VEL
LIN {X 0,Y 390.117,Z 332.888,A -85,B 0,C 180,E1 -11727.929,E2 -11727.929} C_VEL
LIN {X 0,Y 390.023,Z 332.9,A -85,B 0,C 180,E1 -11731.504,E2 -11731.504} C_VEL
LIN {X 0,Y 390.083,Z 332.894,A -85,B 0,C 180,E1 -11735.206,E2 -11735.206} C_VEL
LIN {X 0,Y 390.066,Z 332.896,A -85,B 0,C 180,E1 -11739.217,E2 -11739.217} C_VEL
LIN {X 0,Y 390.041,Z 332.9,A -85,B 0,C 180,E1 -11742.374,E2 -11742.374} C_VEL
LIN {X 0,Y 390.042,Z 332.898,A -85,B 0,C 180,E1 -11745.354,E2 -11745.354} C_VEL
LIN {X 0,Y 390.029,Z 332.9,A -85,B 0,C 180,E1 -11748.186,E2 -11748.186} C_VEL
LIN {X 0,Y 390.09,Z 332.894,A -85,B 0,C 180,E1 -11750.908,E2 -11750.908} C_VEL
LIN {X 0,Y 390.083,Z 332.895,A -85,B 0,C 180,E1 -11754.793,E2 -11754.793} C_VEL
LIN {X 0,Y 390.021,Z 332.905,A -85,B 0,C 180,E1 -11758.495,E2 -11758.495} C_VEL
LIN {X 0,Y 390.114,Z 332.89,A -85,B 0,C 180,E1 -11762.07,E2 -11762.07} C_VEL
LIN {X 0,Y 390.077,Z 332.893,A -85,B 0,C 180,E1 -11765.519,E2 -11765.519} C_VEL
LIN {X 0,Y 390.06,Z 332.897,A -85,B 0,C 180,E1 -11768.878,E2 -11768.878} C_VEL
LIN {X 0,Y 390.125,Z 332.89,A -85,B 0,C 180,E1 -11772.167,E2 -11772.167} C_VEL
LIN {X 0,Y 390.141,Z 332.885,A -85,B 0,C 180,E1 -11775.393,E2 -11775.393} C_VEL
LIN {X 0,Y 390.146,Z 332.888,A -85,B 0,C 180,E1 -11778.571,E2 -11778.571} C_VEL
LIN {X 0,Y 390.341,Z 332.862,A -85,B 0,C 180,E1 -11781.993,E2 -11781.993} C_VEL
LIN {X 0,Y 390.224,Z 332.876,A -85,B 0,C 180,E1 -11784.834,E2 -11784.834} C_VEL
LIN {X 0,Y 390.418,Z 332.852,A -85,B 0,C 180,E1 -11787.937,E2 -11787.937} C_VEL
LIN {X 0,Y 390.548,Z 332.837,A -85,B 0,C 180,E1 -11790,E2 -11790} C_VEL
LIN {X 0,Y 390.313,Z 332.864,A -85,B 0,C 180,E1 -11793.097,E2 -11793.097} C_VEL
LIN {X 0,Y 390.328,Z 332.867,A -85,B 0,C 180,E1 -11796.202,E2 -11796.202} C_VEL
LIN {X 0,Y 390.312,Z 332.868,A -85,B 0,C 180,E1 -11798.282,E2 -11798.282} C_VEL
LIN {X 0,Y 390.168,Z 332.884,A -85,B 0,C 180,E1 -11802.483,E2 -11802.483} C_VEL
LIN {X 0,Y 390.137,Z 332.887,A -85,B 0,C 180,E1 -11805.677,E2 -11805.677} C_VEL
LIN {X 0,Y 390.1,Z 332.891,A -85,B 0,C 180,E1 -11808.977,E2 -11808.977} C_VEL
LIN {X 0,Y 389.406,Z 332.98,A -85,B 0,C 180,E1 -11809.838,E2 -11809.838} C_VEL
LIN {X 0,Y 386.553,Z 333.332,A -85,B 0,C 180,E1 -11811.238,E2 -11811.238} C_VEL
LIN {X 0,Y 384.152,Z 333.634,A -85,B 0,C 180,E1 -11812.369,E2 -11812.369} C_VEL
LIN {X 0,Y 383.12,Z 333.76,A -85,B 0,C 180,E1 -11813.243,E2 -11813.243} C_VEL
LIN {X 0,Y 383.033,Z 333.771,A -85,B 0,C 180,E1 -11813.539,E2 -11813.539} C_VEL
LIN {X 0,Y 383.078,Z 333.769,A -85,B 0,C 180,E1 -11816.124,E2 -11816.124} C_VEL
LIN {X 0,Y 382.99,Z 333.778,A -85,B 0,C 180,E1 -11819.7,E2 -11819.7} C_VEL
LIN {X 0,Y 383.01,Z 333.774,A -85,B 0,C 180,E1 -11823.4,E2 -11823.4} C_VEL
LIN {X 0,Y 383.033,Z 333.774,A -85,B 0,C 180,E1 -11826.166,E2 -11826.166} C_VEL
LIN {X 0,Y 383.009,Z 333.778,A -85,B 0,C 180,E1 -11829.959,E2 -11829.959} C_VEL
LIN {X 0,Y 383.005,Z 333.775,A -85,B 0,C 180,E1 -11832.779,E2 -11832.779} C_VEL
LIN {X 0,Y 382.997,Z 333.779,A -85,B 0,C 180,E1 -11835.79,E2 -11835.79} C_VEL
LIN {X 0,Y 382.988,Z 333.776,A -85,B 0,C 180,E1 -11838.797,E2 -11838.797} C_VEL
LIN {X 0,Y 382.999,Z 333.778,A -85,B 0,C 180,E1 -11842.097,E2 -11842.097} C_VEL
LIN {X 0,Y 383.019,Z 333.773,A -85,B 0,C 180,E1 -11845.333,E2 -11845.333} C_VEL
LIN {X 0,Y 382.984,Z 333.777,A -85,B 0,C 180,E1 -11849.082,E2 -11849.082} C_VEL
LIN {X 0,Y 383.15,Z 333.922,A -85,B 0,C 180,E1 -11852.529,E2 -11852.529} C_VEL
LIN {X 0,Y 388.64,Z 350.477,A -85,B 0,C 180,E1 -11853.14,E2 -11853.14} C_VEL
LIN {X 0,Y 387.273,Z 421.478,A -85,B 0,C 180,E1 -11854.753,E2 -11854.753} C_VEL
LIN {X 0,Y 387.175,Z 434.12,A -85,B 0,C 180,E1 -11855.246,E2 -11855.246} C_VEL
LIN {X 0,Y 386.718,Z 447.83,A -85,B 0,C 180,E1 -11856.007,E2 -11856.007} C_VEL
LIN {X 0,Y 386.267,Z 459.04,A -85,B 0,C 180,E1 -11856.831,E2 -11856.831} C_VEL
LIN {X 0,Y 385.638,Z 471.043,A -85,B 0,C 180,E1 -11857.955,E2 -11857.955} C_VEL
LIN {X 0,Y 385.097,Z 481.317,A -85,B 0,C 180,E1 -11859.154,E2 -11859.154} C_VEL
LIN {X 0,Y 384.409,Z 490.761,A -85,B 0,C 180,E1 -11860.51,E2 -11860.51} C_VEL
LIN {X 0,Y 383.967,Z 498.544,A -85,B 0,C 180,E1 -11861.871,E2 -11861.871} C_VEL
LIN {X 0,Y 383.499,Z 506.128,A -85,B 0,C 180,E1 -11863.498,E2 -11863.498} C_VEL
LIN {X 0,Y 383.1,Z 512.098,A -85,B 0,C 180,E1 -11865.118,E2 -11865.118} C_VEL
LIN {X 0,Y 382.917,Z 516.406,A -85,B 0,C 180,E1 -11866.597,E2 -11866.597} C_VEL
LIN {X 0,Y 382.691,Z 520.246,A -85,B 0,C 180,E1 -11868.346,E2 -11868.346} C_VEL
LIN {X 0,Y 382.631,Z 521.996,A -85,B 0,C 180,E1 -11869.417,E2 -11869.417} C_VEL
LIN {X 0,Y 382.646,Z 523.247,A -85,B 0,C 180,E1 -11870.486,E2 -11870.486} C_VEL
LIN {X 0,Y 382.782,Z 524.471,A -85,B 0,C 180,E1 -11872.509,E2 -11872.509} C_VEL
LIN {X 0,Y 382.86,Z 524.457,A -85,B 0,C 180,E1 -11873.677,E2 -11873.677} C_VEL
LIN {X 0,Y 382.91,Z 524.008,A -85,B 0,C 180,E1 -11874.735,E2 -11874.735} C_VEL
LIN {X 0,Y 382.995,Z 523.162,A -85,B 0,C 180,E1 -11875.791,E2 -11875.791} C_VEL
LIN {X 0,Y 383.262,Z 521.819,A -85,B 0,C 180,E1 -11876.847,E2 -11876.847} C_VEL
LIN {X 0,Y 383.688,Z 518.996,A -85,B 0,C 180,E1 -11878.426,E2 -11878.426} C_VEL
LIN {X 0,Y 384.232,Z 515.089,A -85,B 0,C 180,E1 -11880,E2 -11880} C_VEL
LIN {X 0,Y 384.866,Z 509.996,A -85,B 0,C 180,E1 -11881.57,E2 -11881.57} C_VEL
LIN {X 0,Y 385.61,Z 503.612,A -85,B 0,C 180,E1 -11883.135,E2 -11883.135} C_VEL
LIN {X 0,Y 386.558,Z 495.569,A -85,B 0,C 180,E1 -11884.693,E2 -11884.693} C_VEL
LIN {X 0,Y 387.357,Z 487.35,A -85,B 0,C 180,E1 -11885.989,E2 -11885.989} C_VEL
LIN {X 0,Y 388.32,Z 477.252,A -85,B 0,C 180,E1 -11887.279,E2 -11887.279} C_VEL
LIN {X 0,Y 389.151,Z 465.825,A -85,B 0,C 180,E1 -11888.438,E2 -11888.438} C_VEL
LIN {X 0,Y 389.889,Z 454.575,A -85,B 0,C 180,E1 -11889.337,E2 -11889.337} C_VEL
LIN {X 0,Y 390.418,Z 442.006,A -85,B 0,C 180,E1 -11890.109,E2 -11890.109} C_VEL
LIN {X 0,Y 390.752,Z 428.974,A -85,B 0,C 180,E1 -11890.69,E2 -11890.69} C_VEL
LIN {X 0,Y 391.168,Z 406.325,A -85,B 0,C 180,E1 -11891.301,E2 -11891.301} C_VEL
LIN {X 0,Y 392.963,Z 354.684,A -85,B 0,C 180,E1 -11892.59,E2 -11892.59} C_VEL
LIN {X 0,Y 386.41,Z 340.6,A -85,B 0,C 180,E1 -11893.58,E2 -11893.58} C_VEL
LIN {X 0,Y 383.339,Z 334.823,A -85,B 0,C 180,E1 -11894.045,E2 -11894.045} C_VEL
LIN {X 0,Y 383.121,Z 333.764,A -85,B 0,C 180,E1 -11894.126,E2 -11894.126} C_VEL
LIN {X 0,Y 383.061,Z 333.773,A -85,B 0,C 180,E1 -11897.437,E2 -11897.437} C_VEL
LIN {X 0,Y 383.016,Z 333.776,A -85,B 0,C 180,E1 -11900.64,E2 -11900.64} C_VEL
LIN {X 0,Y 383.011,Z 333.776,A -85,B 0,C 180,E1 -11903.809,E2 -11903.809} C_VEL
LIN {X 0,Y 382.971,Z 333.781,A -85,B 0,C 180,E1 -11907.309,E2 -11907.309} C_VEL
LIN {X 0,Y 382.985,Z 333.779,A -85,B 0,C 180,E1 -11910.919,E2 -11910.919} C_VEL
LIN {X 0,Y 383.015,Z 333.771,A -85,B 0,C 180,E1 -11914.669,E2 -11914.669} C_VEL
LIN {X 0,Y 382.996,Z 333.774,A -85,B 0,C 180,E1 -11917.902,E2 -11917.902} C_VEL
LIN {X 0,Y 382.964,Z 333.777,A -85,B 0,C 180,E1 -11921.351,E2 -11921.351} C_VEL
LIN {X 0,Y 382.992,Z 333.777,A -85,B 0,C 180,E1 -11924.302,E2 -11924.302} C_VEL
LIN {X 0,Y 383.014,Z 333.775,A -85,B 0,C 180,E1 -11927.24,E2 -11927.24} C_VEL
LIN {X 0,Y 382.989,Z 333.779,A -85,B 0,C 180,E1 -11930.419,E2 -11930.419} C_VEL
LIN {X 0,Y 383.028,Z 333.774,A -85,B 0,C 180,E1 -11934.044,E2 -11934.044} C_VEL
LIN {X 0,Y 383.063,Z 333.851,A -85,B 0,C 180,E1 -11937.294,E2 -11937.294} C_VEL
LIN {X 0,Y 386.918,Z 351.432,A -85,B 0,C 180,E1 -11940.678,E2 -11940.678} C_VEL
LIN {X 0,Y 387.843,Z 356.373,A -85,B 0,C 180,E1 -11941.597,E2 -11941.597} C_VEL
LIN {X 0,Y 387.02,Z 367.867,A -85,B 0,C 180,E1 -11943.583,E2 -11943.583} C_VEL
LIN {X 0,Y 385.458,Z 389.082,A -85,B 0,C 180,E1 -11947.204,E2 -11947.204} C_VEL
LIN {X 0,Y 385.059,Z 393.768,A -85,B 0,C 180,E1 -11947.998,E2 -11947.998} C_VEL
LIN {X 0,Y 388.258,Z 417.374,A -85,B 0,C 180,E1 -11948.943,E2 -11948.943} C_VEL
LIN {X 0,Y 390.599,Z 444.111,A -85,B 0,C 180,E1 -11949.873,E2 -11949.873} C_VEL
LIN {X 0,Y 388.678,Z 510.463,A -85,B 0,C 180,E1 -11951.518,E2 -11951.518} C_VEL
LIN {X 0,Y 387.862,Z 524.219,A -85,B 0,C 180,E1 -11952.059,E2 -11952.059} C_VEL
LIN {X 0,Y 386.755,Z 537.748,A -85,B 0,C 180,E1 -11952.825,E2 -11952.825} C_VEL
LIN {X 0,Y 385.724,Z 549.914,A -85,B 0,C 180,E1 -11953.731,E2 -11953.731} C_VEL
LIN {X 0,Y 384.563,Z 562.149,A -85,B 0,C 180,E1 -11954.905,E2 -11954.905} C_VEL
LIN {X 0,Y 383.653,Z 573.121,A -85,B 0,C 180,E1 -11956.223,E2 -11956.223} C_VEL
LIN {X 0,Y 382.975,Z 582.047,A -85,B 0,C 180,E1 -11957.548,E2 -11957.548} C_VEL
LIN {X 0,Y 382.492,Z 590.848,A -85,B 0,C 180,E1 -11959.144,E2 -11959.144} C_VEL
LIN {X 0,Y 382.16,Z 598.006,A -85,B 0,C 180,E1 -11960.74,E2 -11960.74} C_VEL
LIN {X 0,Y 382.114,Z 604.551,A -85,B 0,C 180,E1 -11962.603,E2 -11962.603} C_VEL
LIN {X 0,Y 382.187,Z 610.451,A -85,B 0,C 180,E1 -11964.724,E2 -11964.724} C_VEL
LIN {X 0,Y 382.304,Z 612.735,A -85,B 0,C 180,E1 -11965.783,E2 -11965.783} C_VEL
LIN {X 0,Y 382.326,Z 614.465,A -85,B 0,C 180,E1 -11966.839,E2 -11966.839} C_VEL
LIN {X 0,Y 382.303,Z 615.721,A -85,B 0,C 180,E1 -11967.893,E2 -11967.893} C_VEL
LIN {X 0,Y 382.316,Z 616.541,A -85,B 0,C 180,E1 -11968.947,E2 -11968.947} C_VEL
LIN {X 0,Y 382.353,Z 616.89,A -85,B 0,C 180,E1 -11970,E2 -11970} C_VEL
LIN {X 0,Y 382.288,Z 616.755,A -85,B 0,C 180,E1 -11971.053,E2 -11971.053} C_VEL
LIN {X 0,Y 382.25,Z 616.189,A -85,B 0,C 180,E1 -11972.107,E2 -11972.107} C_VEL
LIN {X 0,Y 382.315,Z 615.2,A -85,B 0,C 180,E1 -11973.161,E2 -11973.161} C_VEL
LIN {X 0,Y 382.247,Z 613.702,A -85,B 0,C 180,E1 -11974.217,E2 -11974.217} C_VEL
LIN {X 0,Y 382.109,Z 610.597,A -85,B 0,C 180,E1 -11975.806,E2 -11975.806} C_VEL
LIN {X 0,Y 382.043,Z 606.389,A -85,B 0,C 180,E1 -11977.398,E2 -11977.398} C_VEL
LIN {X 0,Y 382.114,Z 599.951,A -85,B 0,C 180,E1 -11979.261,E2 -11979.261} C_VEL
LIN {X 0,Y 382.414,Z 592.993,A -85,B 0,C 180,E1 -11980.858,E2 -11980.858} C_VEL
LIN {X 0,Y 382.973,Z 584.376,A -85,B 0,C 180,E1 -11982.452,E2 -11982.452} C_VEL
LIN {X 0,Y 383.802,Z 574.442,A -85,B 0,C 180,E1 -11983.948,E2 -11983.948} C_VEL
LIN {X 0,Y 384.78,Z 564.064,A -85,B 0,C 180,E1 -11985.222,E2 -11985.222} C_VEL
LIN {X 0,Y 385.984,Z 552.165,A -85,B 0,C 180,E1 -11986.393,E2 -11986.393} C_VEL
LIN {X 0,Y 387.256,Z 538.907,A -85,B 0,C 180,E1 -11987.424,E2 -11987.424} C_VEL
LIN {X 0,Y 388.396,Z 525.857,A -85,B 0,C 180,E1 -11988.188,E2 -11988.188} C_VEL
LIN {X 0,Y 389.361,Z 511.681,A -85,B 0,C 180,E1 -11988.789,E2 -11988.789} C_VEL
LIN {X 0,Y 390.038,Z 493.023,A -85,B 0,C 180,E1 -11989.301,E2 -11989.301} C_VEL
LIN {X 0,Y 391.605,Z 442.677,A -85,B 0,C 180,E1 -11990.595,E2 -11990.595} C_VEL
LIN {X 0,Y 389.967,Z 421.508,A -85,B 0,C 180,E1 -11991.354,E2 -11991.354} C_VEL
LIN {X 0,Y 387.629,Z 404.293,A -85,B 0,C 180,E1 -11992.085,E2 -11992.085} C_VEL
LIN {X 0,Y 385.738,Z 393.798,A -85,B 0,C 180,E1 -11992.601,E2 -11992.601} C_VEL
LIN {X 0,Y 387.491,Z 376.478,A -85,B 0,C 180,E1 -11995.804,E2 -11995.804} C_VEL
LIN {X 0,Y 389.47,Z 360.675,A -85,B 0,C 180,E1 -11998.862,E2 -11998.862} C_VEL
LIN {X 0,Y 388.142,Z 352.809,A -85,B 0,C 180,E1 -12000.706,E2 -12000.706} C_VEL
LIN {X 0,Y 385.913,Z 343.701,A -85,B 0,C 180,E1 -12003.116,E2 -12003.116} C_VEL
LIN {X 0,Y 383.551,Z 335.617,A -85,B 0,C 180,E1 -12005.575,E2 -12005.575} C_VEL
LIN {X 0,Y 383.021,Z 333.774,A -85,B 0,C 180,E1 -12006.217,E2 -12006.217} C_VEL
LIN {X 0,Y 382.977,Z 333.783,A -85,B 0,C 180,E1 -12009.962,E2 -12009.962} C_VEL
LIN {X 0,Y 383.008,Z 333.778,A -85,B 0,C 180,E1 -12012.778,E2 -12012.778} C_VEL
LIN {X 0,Y 382.997,Z 333.779,A -85,B 0,C 180,E1 -12015.789,E2 -12015.789} C_VEL
LIN {X 0,Y 382.964,Z 333.782,A -85,B 0,C 180,E1 -12018.8,E2 -12018.8} C_VEL
LIN {X 0,Y 382.994,Z 333.777,A -85,B 0,C 180,E1 -12022.098,E2 -12022.098} C_VEL
LIN {X 0,Y 383.013,Z 333.775,A -85,B 0,C 180,E1 -12025.331,E2 -12025.331} C_VEL
LIN {X 0,Y 382.983,Z 333.78,A -85,B 0,C 180,E1 -12029.081,E2 -12029.081} C_VEL
LIN {X 0,Y 382.968,Z 333.781,A -85,B 0,C 180,E1 -12032.691,E2 -12032.691} C_VEL
LIN {X 0,Y 383.009,Z 333.78,A -85,B 0,C 180,E1 -12036.191,E2 -12036.191} C_VEL
LIN {X 0,Y 383.048,Z 333.773,A -85,B 0,C 180,E1 -12039.486,E2 -12039.486} C_VEL
LIN {X 0,Y 384.093,Z 336.729,A -85,B 0,C 180,E1 -12039.713,E2 -12039.713} C_VEL
LIN {X 0,Y 385.346,Z 338.794,A -85,B 0,C 180,E1 -12039.919,E2 -12039.919} C_VEL
LIN {X 0,Y 391.423,Z 350.39,A -85,B 0,C 180,E1 -12040.903,E2 -12040.903} C_VEL
LIN {X 0,Y 393.84,Z 355.728,A -85,B 0,C 180,E1 -12041.295,E2 -12041.295} C_VEL
LIN {X 0,Y 391.26,Z 421.184,A -85,B 0,C 180,E1 -12043.028,E2 -12043.028} C_VEL
LIN {X 0,Y 391.057,Z 434.456,A -85,B 0,C 180,E1 -12043.49,E2 -12043.49} C_VEL
LIN {X 0,Y 390.627,Z 447.29,A -85,B 0,C 180,E1 -12044.142,E2 -12044.142} C_VEL
LIN {X 0,Y 389.964,Z 459.587,A -85,B 0,C 180,E1 -12044.985,E2 -12044.985} C_VEL
LIN {X 0,Y 389.118,Z 471.29,A -85,B 0,C 180,E1 -12046.02,E2 -12046.02} C_VEL
LIN {X 0,Y 388.252,Z 481.723,A -85,B 0,C 180,E1 -12047.188,E2 -12047.188} C_VEL
LIN {X 0,Y 387.327,Z 491.116,A -85,B 0,C 180,E1 -12048.486,E2 -12048.486} C_VEL
LIN {X 0,Y 386.458,Z 498.824,A -85,B 0,C 180,E1 -12049.786,E2 -12049.786} C_VEL
LIN {X 0,Y 385.492,Z 506.376,A -85,B 0,C 180,E1 -12051.349,E2 -12051.349} C_VEL
LIN {X 0,Y 384.905,Z 511.44,A -85,B 0,C 180,E1 -12052.656,E2 -12052.656} C_VEL
LIN {X 0,Y 384.239,Z 516.321,A -85,B 0,C 180,E1 -12054.226,E2 -12054.226} C_VEL
LIN {X 0,Y 383.69,Z 520.037,A -85,B 0,C 180,E1 -12055.798,E2 -12055.798} C_VEL
LIN {X 0,Y 383.395,Z 521.899,A -85,B 0,C 180,E1 -12056.847,E2 -12056.847} C_VEL
LIN {X 0,Y 383.249,Z 523.316,A -85,B 0,C 180,E1 -12057.898,E2 -12057.898} C_VEL
LIN {X 0,Y 383.085,Z 524.317,A -85,B 0,C 180,E1 -12058.948,E2 -12058.948} C_VEL
LIN {X 0,Y 382.963,Z 524.853,A -85,B 0,C 180,E1 -12060,E2 -12060} C_VEL
LIN {X 0,Y 382.805,Z 524.993,A -85,B 0,C 180,E1 -12061.051,E2 -12061.051} C_VEL
LIN {X 0,Y 382.501,Z 524.751,A -85,B 0,C 180,E1 -12062.105,E2 -12062.105} C_VEL
LIN {X 0,Y 382.516,Z 524.015,A -85,B 0,C 180,E1 -12063.159,E2 -12063.159} C_VEL
LIN {X 0,Y 382.678,Z 522.841,A -85,B 0,C 180,E1 -12064.212,E2 -12064.212} C_VEL
LIN {X 0,Y 382.85,Z 520.289,A -85,B 0,C 180,E1 -12065.794,E2 -12065.794} C_VEL
LIN {X 0,Y 382.942,Z 515.953,A -85,B 0,C 180,E1 -12067.673,E2 -12067.673} C_VEL
LIN {X 0,Y 383.256,Z 510.128,A -85,B 0,C 180,E1 -12069.499,E2 -12069.499} C_VEL
LIN {X 0,Y 383.605,Z 503.638,A -85,B 0,C 180,E1 -12071.091,E2 -12071.091} C_VEL
LIN {X 0,Y 384.12,Z 495.56,A -85,B 0,C 180,E1 -12072.682,E2 -12072.682} C_VEL
LIN {X 0,Y 384.661,Z 486.782,A -85,B 0,C 180,E1 -12074.077,E2 -12074.077} C_VEL
LIN {X 0,Y 385.152,Z 477.107,A -85,B 0,C 180,E1 -12075.342,E2 -12075.342} C_VEL
LIN {X 0,Y 385.768,Z 465.812,A -85,B 0,C 180,E1 -12076.538,E2 -12076.538} C_VEL
LIN {X 0,Y 386.311,Z 452.978,A -85,B 0,C 180,E1 -12077.604,E2 -12077.604} C_VEL
LIN {X 0,Y 386.868,Z 440.442,A -85,B 0,C 180,E1 -12078.399,E2 -12078.399} C_VEL
LIN {X 0,Y 387.115,Z 426.533,A -85,B 0,C 180,E1 -12079.039,E2 -12079.039} C_VEL
LIN {X 0,Y 387.251,Z 412.495,A -85,B 0,C 180,E1 -12079.453,E2 -12079.453} C_VEL
LIN {X 0,Y 388.37,Z 349.881,A -85,B 0,C 180,E1 -12080.897,E2 -12080.897} C_VEL
LIN {X 0,Y 383.027,Z 333.772,A -85,B 0,C 180,E1 -12081.498,E2 -12081.498} C_VEL
LIN {X 0,Y 383.053,Z 333.772,A -85,B 0,C 180,E1 -12084.96,E2 -12084.96} C_VEL
LIN {X 0,Y 383.04,Z 333.772,A -85,B 0,C 180,E1 -12088.492,E2 -12088.492} C_VEL
LIN {X 0,Y 383.008,Z 333.774,A -85,B 0,C 180,E1 -12092.149,E2 -12092.149} C_VEL
LIN {X 0,Y 383.017,Z 333.777,A -85,B 0,C 180,E1 -12094.667,E2 -12094.667} C_VEL
LIN {X 0,Y 382.997,Z 333.775,A -85,B 0,C 180,E1 -12097.903,E2 -12097.903} C_VEL
LIN {X 0,Y 382.982,Z 333.778,A -85,B 0,C 180,E1 -12101.347,E2 -12101.347} C_VEL
LIN {X 0,Y 382.994,Z 333.777,A -85,B 0,C 180,E1 -12104.303,E2 -12104.303} C_VEL
LIN {X 0,Y 383.008,Z 333.775,A -85,B 0,C 180,E1 -12107.24,E2 -12107.24} C_VEL
LIN {X 0,Y 383.014,Z 333.776,A -85,B 0,C 180,E1 -12110.413,E2 -12110.413} C_VEL
LIN {X 0,Y 383.024,Z 333.772,A -85,B 0,C 180,E1 -12114.044,E2 -12114.044} C_VEL
LIN {X 0,Y 382.984,Z 333.776,A -85,B 0,C 180,E1 -12117.578,E2 -12117.578} C_VEL
LIN {X 0,Y 382.99,Z 333.779,A -85,B 0,C 180,E1 -12120.3,E2 -12120.3} C_VEL
LIN {X 0,Y 383.078,Z 333.766,A -85,B 0,C 180,E1 -12124.021,E2 -12124.021} C_VEL
LIN {X 0,Y 383.01,Z 333.773,A -85,B 0,C 180,E1 -12127.335,E2 -12127.335} C_VEL
LIN {X 0,Y 383.058,Z 333.77,A -85,B 0,C 180,E1 -12130.716,E2 -12130.716} C_VEL
LIN {X 0,Y 383.078,Z 333.766,A -85,B 0,C 180,E1 -12134.027,E2 -12134.027} C_VEL
LIN {X 0,Y 383.133,Z 333.758,A -85,B 0,C 180,E1 -12137.284,E2 -12137.284} C_VEL
LIN {X 0,Y 383.152,Z 333.759,A -85,B 0,C 180,E1 -12140.498,E2 -12140.498} C_VEL
LIN {X 0,Y 383.271,Z 333.744,A -85,B 0,C 180,E1 -12142.625,E2 -12142.625} C_VEL
LIN {X 0,Y 383.197,Z 333.752,A -85,B 0,C 180,E1 -12144.739,E2 -12144.739} C_VEL
LIN {X 0,Y 383.385,Z 333.728,A -85,B 0,C 180,E1 -12147.899,E2 -12147.899} C_VEL
LIN {X 0,Y 383.517,Z 333.713,A -85,B 0,C 180,E1 -12150,E2 -12150} C_VEL
LIN {X 0,Y 383.249,Z 333.744,A -85,B 0,C 180,E1 -12153.154,E2 -12153.154} C_VEL
LIN {X 0,Y 383.285,Z 333.743,A -85,B 0,C 180,E1 -12156.317,E2 -12156.317} C_VEL
LIN {X 0,Y 383.257,Z 333.746,A -85,B 0,C 180,E1 -12158.436,E2 -12158.436} C_VEL
LIN {X 0,Y 383.095,Z 333.763,A -85,B 0,C 180,E1 -12161.642,E2 -12161.642} C_VEL
LIN {X 0,Y 383.108,Z 333.762,A -85,B 0,C 180,E1 -12164.882,E2 -12164.882} C_VEL
LIN {X 0,Y 383.087,Z 333.768,A -85,B 0,C 180,E1 -12168.173,E2 -12168.173} C_VEL
LIN {X 0,Y 382.991,Z 333.776,A -85,B 0,C 180,E1 -12171.531,E2 -12171.531} C_VEL
LIN {X 0,Y 383.033,Z 333.771,A -85,B 0,C 180,E1 -12173.539,E2 -12173.539} C_VEL
LIN {X 0,Y 382.358,Z 333.859,A -85,B 0,C 180,E1 -12174.418,E2 -12174.418} C_VEL
LIN {X 0,Y 379.499,Z 334.217,A -85,B 0,C 180,E1 -12175.846,E2 -12175.846} C_VEL
LIN {X 0,Y 377.087,Z 334.515,A -85,B 0,C 180,E1 -12177,E2 -12177} C_VEL
LIN {X 0,Y 376.056,Z 334.643,A -85,B 0,C 180,E1 -12177.893,E2 -12177.893} C_VEL
LIN {X 0,Y 375.975,Z 334.651,A -85,B 0,C 180,E1 -12178.196,E2 -12178.196} C_VEL
LIN {X 0,Y 375.957,Z 334.653,A -85,B 0,C 180,E1 -12181.563,E2 -12181.563} C_VEL
LIN {X 0,Y 375.957,Z 334.652,A -85,B 0,C 180,E1 -12185.416,E2 -12185.416} C_VEL
LIN {X 0,Y 375.976,Z 334.652,A -85,B 0,C 180,E1 -12188.272,E2 -12188.272} C_VEL
LIN {X 0,Y 375.934,Z 334.657,A -85,B 0,C 180,E1 -12191.602,E2 -12191.602} C_VEL
LIN {X 0,Y 375.927,Z 334.656,A -85,B 0,C 180,E1 -12195.269,E2 -12195.269} C_VEL
LIN {X 0,Y 375.934,Z 334.657,A -85,B 0,C 180,E1 -12198.4,E2 -12198.4} C_VEL
LIN {X 0,Y 375.973,Z 334.654,A -85,B 0,C 180,E1 -12201.731,E2 -12201.731} C_VEL
LIN {X 0,Y 375.981,Z 334.65,A -85,B 0,C 180,E1 -12205.333,E2 -12205.333} C_VEL
LIN {X 0,Y 375.959,Z 334.653,A -85,B 0,C 180,E1 -12208.439,E2 -12208.439} C_VEL
LIN {X 0,Y 376.065,Z 334.641,A -85,B 0,C 180,E1 -12212.232,E2 -12212.232} C_VEL
LIN {X 0,Y 381.683,Z 351.691,A -85,B 0,C 180,E1 -12212.895,E2 -12212.895} C_VEL
LIN {X 0,Y 380.369,Z 421.631,A -85,B 0,C 180,E1 -12214.523,E2 -12214.523} C_VEL
LIN {X 0,Y 380.214,Z 435.048,A -85,B 0,C 180,E1 -12215.052,E2 -12215.052} C_VEL
LIN {X 0,Y 379.751,Z 448.739,A -85,B 0,C 180,E1 -12215.829,E2 -12215.829} C_VEL
LIN {X 0,Y 379.291,Z 459.914,A -85,B 0,C 180,E1 -12216.668,E2 -12216.668} C_VEL
LIN {X 0,Y 378.671,Z 471.599,A -85,B 0,C 180,E1 -12217.781,E2 -12217.781} C_VEL
LIN {X 0,Y 378.098,Z 482.18,A -85,B 0,C 180,E1 -12219.035,E2 -12219.035} C_VEL
LIN {X 0,Y 377.401,Z 491.627,A -85,B 0,C 180,E1 -12220.416,E2 -12220.416} C_VEL
LIN {X 0,Y 376.854,Z 500.493,A -85,B 0,C 180,E1 -12222.011,E2 -12222.011} C_VEL
LIN {X 0,Y 376.367,Z 508.078,A -85,B 0,C 180,E1 -12223.734,E2 -12223.734} C_VEL
LIN {X 0,Y 376.012,Z 513.849,A -85,B 0,C 180,E1 -12225.385,E2 -12225.385} C_VEL
LIN {X 0,Y 375.815,Z 518.331,A -85,B 0,C 180,E1 -12227.032,E2 -12227.032} C_VEL
LIN {X 0,Y 375.684,Z 520.647,A -85,B 0,C 180,E1 -12228.125,E2 -12228.125} C_VEL
LIN {X 0,Y 375.588,Z 522.492,A -85,B 0,C 180,E1 -12229.216,E2 -12229.216} C_VEL
LIN {X 0,Y 375.588,Z 523.907,A -85,B 0,C 180,E1 -12230.305,E2 -12230.305} C_VEL
LIN {X 0,Y 375.651,Z 524.827,A -85,B 0,C 180,E1 -12231.393,E2 -12231.393} C_VEL
LIN {X 0,Y 375.742,Z 525.339,A -85,B 0,C 180,E1 -12232.477,E2 -12232.477} C_VEL
LIN {X 0,Y 375.835,Z 525.441,A -85,B 0,C 180,E1 -12233.558,E2 -12233.558} C_VEL
LIN {X 0,Y 375.886,Z 525.078,A -85,B 0,C 180,E1 -12234.636,E2 -12234.636} C_VEL
LIN {X 0,Y 375.963,Z 524.312,A -85,B 0,C 180,E1 -12235.712,E2 -12235.712} C_VEL
LIN {X 0,Y 376.25,Z 523.108,A -85,B 0,C 180,E1 -12236.788,E2 -12236.788} C_VEL
LIN {X 0,Y 376.687,Z 520.452,A -85,B 0,C 180,E1 -12238.397,E2 -12238.397} C_VEL
LIN {X 0,Y 377.254,Z 516.739,A -85,B 0,C 180,E1 -12240.001,E2 -12240.001} C_VEL
LIN {X 0,Y 377.935,Z 511.85,A -85,B 0,C 180,E1 -12241.599,E2 -12241.599} C_VEL
LIN {X 0,Y 378.718,Z 505.654,A -85,B 0,C 180,E1 -12243.192,E2 -12243.192} C_VEL
LIN {X 0,Y 379.727,Z 497.9,A -85,B 0,C 180,E1 -12244.778,E2 -12244.778} C_VEL
LIN {X 0,Y 380.568,Z 489.95,A -85,B 0,C 180,E1 -12246.096,E2 -12246.096} C_VEL
LIN {X 0,Y 381.555,Z 480.189,A -85,B 0,C 180,E1 -12247.409,E2 -12247.409} C_VEL
LIN {X 0,Y 382.428,Z 469.446,A -85,B 0,C 180,E1 -12248.588,E2 -12248.588} C_VEL
LIN {X 0,Y 383.342,Z 457.15,A -85,B 0,C 180,E1 -12249.631,E2 -12249.631} C_VEL
LIN {X 0,Y 383.936,Z 445.243,A -85,B 0,C 180,E1 -12250.415,E2 -12250.415} C_VEL
LIN {X 0,Y 384.343,Z 431.4,A -85,B 0,C 180,E1 -12251.07,E2 -12251.07} C_VEL
LIN {X 0,Y 384.579,Z 414.835,A -85,B 0,C 180,E1 -12251.564,E2 -12251.564} C_VEL
LIN {X 0,Y 386.723,Z 356.652,A -85,B 0,C 180,E1 -12253.065,E2 -12253.065} C_VEL
LIN {X 0,Y 380.693,Z 343.97,A -85,B 0,C 180,E1 -12254.008,E2 -12254.008} C_VEL
LIN {X 0,Y 377.126,Z 337.594,A -85,B 0,C 180,E1 -12254.576,E2 -12254.576} C_VEL
LIN {X 0,Y 376.075,Z 334.639,A -85,B 0,C 180,E1 -12254.797,E2 -12254.797} C_VEL
LIN {X 0,Y 375.982,Z 334.653,A -85,B 0,C 180,E1 -12258.529,E2 -12258.529} C_VEL
LIN {X 0,Y 375.954,Z 334.661,A -85,B 0,C 180,E1 -12261.955,E2 -12261.955} C_VEL
LIN {X 0,Y 375.961,Z 334.659,A -85,B 0,C 180,E1 -12264.284,E2 -12264.284} C_VEL
LIN {X 0,Y 375.92,Z 334.66,A -85,B 0,C 180,E1 -12267.865,E2 -12267.865} C_VEL
LIN {X 0,Y 375.96,Z 334.655,A -85,B 0,C 180,E1 -12271.562,E2 -12271.562} C_VEL
LIN {X 0,Y 375.952,Z 334.65,A -85,B 0,C 180,E1 -12275.417,E2 -12275.417} C_VEL
LIN {X 0,Y 375.938,Z 334.653,A -85,B 0,C 180,E1 -12278.263,E2 -12278.263} C_VEL
LIN {X 0,Y 375.919,Z 334.655,A -85,B 0,C 180,E1 -12281.597,E2 -12281.597} C_VEL
LIN {X 0,Y 375.925,Z 334.657,A -85,B 0,C 180,E1 -12284.73,E2 -12284.73} C_VEL
LIN {X 0,Y 375.929,Z 334.659,A -85,B 0,C 180,E1 -12287.699,E2 -12287.699} C_VEL
LIN {X 0,Y 375.938,Z 334.657,A -85,B 0,C 180,E1 -12290.534,E2 -12290.534} C_VEL
LIN {X 0,Y 375.966,Z 334.655,A -85,B 0,C 180,E1 -12293.496,E2 -12293.496} C_VEL
LIN {X 0,Y 376.018,Z 334.793,A -85,B 0,C 180,E1 -12297.058,E2 -12297.058} C_VEL
LIN {X 0,Y 379.785,Z 351.967,A -85,B 0,C 180,E1 -12300.43,E2 -12300.43} C_VEL
LIN {X 0,Y 380.882,Z 358.509,A -85,B 0,C 180,E1 -12301.661,E2 -12301.661} C_VEL
LIN {X 0,Y 379.161,Z 379.127,A -85,B 0,C 180,E1 -12305.265,E2 -12305.265} C_VEL
LIN {X 0,Y 378.31,Z 390.782,A -85,B 0,C 180,E1 -12307.29,E2 -12307.29} C_VEL
LIN {X 0,Y 381.843,Z 416.938,A -85,B 0,C 180,E1 -12308.421,E2 -12308.421} C_VEL
LIN {X 0,Y 384.224,Z 444.645,A -85,B 0,C 180,E1 -12309.415,E2 -12309.415} C_VEL
LIN {X 0,Y 382.179,Z 509.615,A -85,B 0,C 180,E1 -12311.088,E2 -12311.088} C_VEL
LIN {X 0,Y 381.359,Z 522.574,A -85,B 0,C 180,E1 -12311.603,E2 -12311.603} C_VEL
LIN {X 0,Y 380.398,Z 534.308,A -85,B 0,C 180,E1 -12312.251,E2 -12312.251} C_VEL
LIN {X 0,Y 379.211,Z 546.859,A -85,B 0,C 180,E1 -12313.167,E2 -12313.167} C_VEL
LIN {X 0,Y 378.099,Z 558.275,A -85,B 0,C 180,E1 -12314.226,E2 -12314.226} C_VEL
LIN {X 0,Y 377.121,Z 568.667,A -85,B 0,C 180,E1 -12315.428,E2 -12315.428} C_VEL
LIN {X 0,Y 376.34,Z 578.465,A -85,B 0,C 180,E1 -12316.813,E2 -12316.813} C_VEL
LIN {X 0,Y 375.611,Z 587.617,A -85,B 0,C 180,E1 -12318.396,E2 -12318.396} C_VEL
LIN {X 0,Y 375.187,Z 595.158,A -85,B 0,C 180,E1 -12320.022,E2 -12320.022} C_VEL
LIN {X 0,Y 375.032,Z 602.166,A -85,B 0,C 180,E1 -12321.92,E2 -12321.92} C_VEL
LIN {X 0,Y 375.101,Z 606.792,A -85,B 0,C 180,E1 -12323.545,E2 -12323.545} C_VEL
LIN {X 0,Y 375.259,Z 611.622,A -85,B 0,C 180,E1 -12325.704,E2 -12325.704} C_VEL
LIN {X 0,Y 375.282,Z 613.421,A -85,B 0,C 180,E1 -12326.779,E2 -12326.779} C_VEL
LIN {X 0,Y 375.265,Z 614.709,A -85,B 0,C 180,E1 -12327.853,E2 -12327.853} C_VEL
LIN {X 0,Y 375.279,Z 615.558,A -85,B 0,C 180,E1 -12328.927,E2 -12328.927} C_VEL
LIN {X 0,Y 375.313,Z 615.963,A -85,B 0,C 180,E1 -12330,E2 -12330} C_VEL
LIN {X 0,Y 375.24,Z 615.856,A -85,B 0,C 180,E1 -12331.073,E2 -12331.073} C_VEL
LIN {X 0,Y 375.199,Z 615.313,A -85,B 0,C 180,E1 -12332.147,E2 -12332.147} C_VEL
LIN {X 0,Y 375.268,Z 614.351,A -85,B 0,C 180,E1 -12333.221,E2 -12333.221} C_VEL
LIN {X 0,Y 375.163,Z 612.897,A -85,B 0,C 180,E1 -12334.297,E2 -12334.297} C_VEL
LIN {X 0,Y 375.017,Z 609.842,A -85,B 0,C 180,E1 -12335.916,E2 -12335.916} C_VEL
LIN {X 0,Y 374.968,Z 605.686,A -85,B 0,C 180,E1 -12337.539,E2 -12337.539} C_VEL
LIN {X 0,Y 375.053,Z 599.31,A -85,B 0,C 180,E1 -12339.437,E2 -12339.437} C_VEL
LIN {X 0,Y 375.386,Z 592.418,A -85,B 0,C 180,E1 -12341.064,E2 -12341.064} C_VEL
LIN {X 0,Y 376.002,Z 583.94,A -85,B 0,C 180,E1 -12342.687,E2 -12342.687} C_VEL
LIN {X 0,Y 376.937,Z 573.643,A -85,B 0,C 180,E1 -12344.275,E2 -12344.275} C_VEL
LIN {X 0,Y 378.027,Z 562.749,A -85,B 0,C 180,E1 -12345.639,E2 -12345.639} C_VEL
LIN {X 0,Y 379.352,Z 550.825,A -85,B 0,C 180,E1 -12346.826,E2 -12346.826} C_VEL
LIN {X 0,Y 380.525,Z 539.41,A -85,B 0,C 180,E1 -12347.743,E2 -12347.743} C_VEL
LIN {X 0,Y 381.698,Z 526.984,A -85,B 0,C 180,E1 -12348.519,E2 -12348.519} C_VEL
LIN {X 0,Y 382.842,Z 512.177,A -85,B 0,C 180,E1 -12349.191,E2 -12349.191} C_VEL
LIN {X 0,Y 383.483,Z 497.156,A -85,B 0,C 180,E1 -12349.644,E2 -12349.644} C_VEL
LIN {X 0,Y 385.331,Z 443.657,A -85,B 0,C 180,E1 -12351.06,E2 -12351.06} C_VEL
LIN {X 0,Y 383.82,Z 422.816,A -85,B 0,C 180,E1 -12351.835,E2 -12351.835} C_VEL
LIN {X 0,Y 381.57,Z 405.988,A -85,B 0,C 180,E1 -12352.581,E2 -12352.581} C_VEL
LIN {X 0,Y 379.17,Z 392.27,A -85,B 0,C 180,E1 -12353.304,E2 -12353.304} C_VEL
LIN {X 0,Y 381.1,Z 375.199,A -85,B 0,C 180,E1 -12356.564,E2 -12356.564} C_VEL
LIN {X 0,Y 382.78,Z 362.459,A -85,B 0,C 180,E1 -12359.114,E2 -12359.114} C_VEL
LIN {X 0,Y 381.41,Z 354.478,A -85,B 0,C 180,E1 -12361.06,E2 -12361.06} C_VEL
LIN {X 0,Y 379.214,Z 345.668,A -85,B 0,C 180,E1 -12363.489,E2 -12363.489} C_VEL
LIN {X 0,Y 376.928,Z 337.912,A -85,B 0,C 180,E1 -12365.968,E2 -12365.968} C_VEL
LIN {X 0,Y 375.962,Z 334.654,A -85,B 0,C 180,E1 -12367.159,E2 -12367.159} C_VEL
LIN {X 0,Y 375.917,Z 334.662,A -85,B 0,C 180,E1 -12370.87,E2 -12370.87} C_VEL
LIN {X 0,Y 375.931,Z 334.659,A -85,B 0,C 180,E1 -12373.766,E2 -12373.766} C_VEL
LIN {X 0,Y 375.936,Z 334.657,A -85,B 0,C 180,E1 -12376.81,E2 -12376.81} C_VEL
LIN {X 0,Y 375.936,Z 334.656,A -85,B 0,C 180,E1 -12380.533,E2 -12380.533} C_VEL
LIN {X 0,Y 375.959,Z 334.652,A -85,B 0,C 180,E1 -12383.497,E2 -12383.497} C_VEL
LIN {X 0,Y 375.959,Z 334.654,A -85,B 0,C 180,E1 -12385.888,E2 -12385.888} C_VEL
LIN {X 0,Y 375.963,Z 334.655,A -85,B 0,C 180,E1 -12389.687,E2 -12389.687} C_VEL
LIN {X 0,Y 375.918,Z 334.662,A -85,B 0,C 180,E1 -12392.135,E2 -12392.135} C_VEL
LIN {X 0,Y 375.937,Z 334.659,A -85,B 0,C 180,E1 -12394.533,E2 -12394.533} C_VEL
LIN {X 0,Y 375.972,Z 334.656,A -85,B 0,C 180,E1 -12396.886,E2 -12396.886} C_VEL
LIN {X 0,Y 375.966,Z 334.763,A -85,B 0,C 180,E1 -12398.728,E2 -12398.728} C_VEL
LIN {X 0,Y 376.993,Z 337.57,A -85,B 0,C 180,E1 -12398.952,E2 -12398.952} C_VEL
LIN {X 0,Y 378.384,Z 339.579,A -85,B 0,C 180,E1 -12399.187,E2 -12399.187} C_VEL
LIN {X 0,Y 384.967,Z 352.007,A -85,B 0,C 180,E1 -12400.33,E2 -12400.33} C_VEL
LIN {X 0,Y 387.636,Z 357.677,A -85,B 0,C 180,E1 -12400.784,E2 -12400.784} C_VEL
LIN {X 0,Y 384.976,Z 421.38,A -85,B 0,C 180,E1 -12402.537,E2 -12402.537} C_VEL
LIN {X 0,Y 384.758,Z 434.83,A -85,B 0,C 180,E1 -12403.006,E2 -12403.006} C_VEL
LIN {X 0,Y 384.235,Z 448.875,A -85,B 0,C 180,E1 -12403.735,E2 -12403.735} C_VEL
LIN {X 0,Y 383.542,Z 460.964,A -85,B 0,C 180,E1 -12404.591,E2 -12404.591} C_VEL
LIN {X 0,Y 382.635,Z 472.563,A -85,B 0,C 180,E1 -12405.643,E2 -12405.643} C_VEL
LIN {X 0,Y 381.695,Z 482.932,A -85,B 0,C 180,E1 -12406.829,E2 -12406.829} C_VEL
LIN {X 0,Y 380.782,Z 491.444,A -85,B 0,C 180,E1 -12408.018,E2 -12408.018} C_VEL
LIN {X 0,Y 379.687,Z 500.655,A -85,B 0,C 180,E1 -12409.602,E2 -12409.602} C_VEL
LIN {X 0,Y 378.671,Z 508,A -85,B 0,C 180,E1 -12411.192,E2 -12411.192} C_VEL
LIN {X 0,Y 377.772,Z 514.675,A -85,B 0,C 180,E1 -12413.054,E2 -12413.054} C_VEL
LIN {X 0,Y 377.089,Z 519.049,A -85,B 0,C 180,E1 -12414.652,E2 -12414.652} C_VEL
LIN {X 0,Y 376.724,Z 521.312,A -85,B 0,C 180,E1 -12415.72,E2 -12415.72} C_VEL
LIN {X 0,Y 376.411,Z 523.114,A -85,B 0,C 180,E1 -12416.788,E2 -12416.788} C_VEL
LIN {X 0,Y 376.249,Z 524.473,A -85,B 0,C 180,E1 -12417.859,E2 -12417.859} C_VEL
LIN {X 0,Y 376.07,Z 525.376,A -85,B 0,C 180,E1 -12418.929,E2 -12418.929} C_VEL
LIN {X 0,Y 375.949,Z 525.854,A -85,B 0,C 180,E1 -12419.999,E2 -12419.999} C_VEL
LIN {X 0,Y 375.771,Z 525.94,A -85,B 0,C 180,E1 -12421.071,E2 -12421.071} C_VEL
LIN {X 0,Y 375.457,Z 525.615,A -85,B 0,C 180,E1 -12422.145,E2 -12422.145} C_VEL
LIN {X 0,Y 375.471,Z 524.799,A -85,B 0,C 180,E1 -12423.219,E2 -12423.219} C_VEL
LIN {X 0,Y 375.649,Z 523.563,A -85,B 0,C 180,E1 -12424.291,E2 -12424.291} C_VEL
LIN {X 0,Y 375.819,Z 520.896,A -85,B 0,C 180,E1 -12425.903,E2 -12425.903} C_VEL
LIN {X 0,Y 375.906,Z 516.635,A -85,B 0,C 180,E1 -12427.735,E2 -12427.735} C_VEL
LIN {X 0,Y 376.141,Z 512.329,A -85,B 0,C 180,E1 -12429.138,E2 -12429.138} C_VEL
LIN {X 0,Y 376.484,Z 506.153,A -85,B 0,C 180,E1 -12430.758,E2 -12430.758} C_VEL
LIN {X 0,Y 376.957,Z 498.404,A -85,B 0,C 180,E1 -12432.38,E2 -12432.38} C_VEL
LIN {X 0,Y 377.576,Z 488.779,A -85,B 0,C 180,E1 -12434.003,E2 -12434.003} C_VEL
LIN {X 0,Y 378.1,Z 478.754,A -85,B 0,C 180,E1 -12435.359,E2 -12435.359} C_VEL
LIN {X 0,Y 378.679,Z 468.991,A -85,B 0,C 180,E1 -12436.44,E2 -12436.44} C_VEL
LIN {X 0,Y 379.174,Z 456.883,A -85,B 0,C 180,E1 -12437.529,E2 -12437.529} C_VEL
LIN {X 0,Y 379.777,Z 444.117,A -85,B 0,C 180,E1 -12438.406,E2 -12438.406} C_VEL
LIN {X 0,Y 380.119,Z 430.82,A -85,B 0,C 180,E1 -12439.088,E2 -12439.088} C_VEL
LIN {X 0,Y 380.247,Z 416.535,A -85,B 0,C 180,E1 -12439.572,E2 -12439.572} C_VEL
LIN {X 0,Y 381.499,Z 351.381,A -85,B 0,C 180,E1 -12441.118,E2 -12441.118} C_VEL
LIN {X 0,Y 375.964,Z 334.652,A -85,B 0,C 180,E1 -12441.778,E2 -12441.778} C_VEL
LIN {X 0,Y 375.994,Z 334.648,A -85,B 0,C 180,E1 -12444.281,E2 -12444.281} C_VEL
LIN {X 0,Y 376.02,Z 334.648,A -85,B 0,C 180,E1 -12446.651,E2 -12446.651} C_VEL
LIN {X 0,Y 375.97,Z 334.653,A -85,B 0,C 180,E1 -12449.079,E2 -12449.079} C_VEL
LIN {X 0,Y 375.948,Z 334.658,A -85,B 0,C 180,E1 -12452.828,E2 -12452.828} C_VEL
LIN {X 0,Y 375.956,Z 334.653,A -85,B 0,C 180,E1 -12455.415,E2 -12455.415} C_VEL
LIN {X 0,Y 375.971,Z 334.651,A -85,B 0,C 180,E1 -12458.27,E2 -12458.27} C_VEL
LIN {X 0,Y 375.932,Z 334.655,A -85,B 0,C 180,E1 -12461.6,E2 -12461.6} C_VEL
LIN {X 0,Y 375.925,Z 334.657,A -85,B 0,C 180,E1 -12465.268,E2 -12465.268} C_VEL
LIN {X 0,Y 375.933,Z 334.658,A -85,B 0,C 180,E1 -12468.399,E2 -12468.399} C_VEL
LIN {X 0,Y 375.974,Z 334.649,A -85,B 0,C 180,E1 -12471.729,E2 -12471.729} C_VEL
LIN {X 0,Y 375.978,Z 334.65,A -85,B 0,C 180,E1 -12475.332,E2 -12475.332} C_VEL
LIN {X 0,Y 375.955,Z 334.656,A -85,B 0,C 180,E1 -12478.438,E2 -12478.438} C_VEL
LIN {X 0,Y 375.98,Z 334.651,A -85,B 0,C 180,E1 -12482.14,E2 -12482.14} C_VEL
LIN {X 0,Y 376.004,Z 334.651,A -85,B 0,C 180,E1 -12484.539,E2 -12484.539} C_VEL
LIN {X 0,Y 375.965,Z 334.652,A -85,B 0,C 180,E1 -12488.046,E2 -12488.046} C_VEL
LIN {X 0,Y 376.006,Z 334.645,A -85,B 0,C 180,E1 -12491.473,E2 -12491.473} C_VEL
LIN {X 0,Y 376.055,Z 334.642,A -85,B 0,C 180,E1 -12494.833,E2 -12494.833} C_VEL
LIN {X 0,Y 376.048,Z 334.643,A -85,B 0,C 180,E1 -12498.137,E2 -12498.137} C_VEL
LIN {X 0,Y 376.255,Z 334.616,A -85,B 0,C 180,E1 -12501.877,E2 -12501.877} C_VEL
LIN {X 0,Y 376.169,Z 334.628,A -85,B 0,C 180,E1 -12504.64,E2 -12504.64} C_VEL
LIN {X 0,Y 376.351,Z 334.604,A -85,B 0,C 180,E1 -12507.86,E2 -12507.86} C_VEL
LIN {X 0,Y 376.486,Z 334.588,A -85,B 0,C 180,E1 -12510,E2 -12510} C_VEL
LIN {X 0,Y 376.187,Z 334.623,A -85,B 0,C 180,E1 -12513.213,E2 -12513.213} C_VEL
LIN {X 0,Y 376.244,Z 334.62,A -85,B 0,C 180,E1 -12516.435,E2 -12516.435} C_VEL
LIN {X 0,Y 376.203,Z 334.624,A -85,B 0,C 180,E1 -12518.595,E2 -12518.595} C_VEL
LIN {X 0,Y 376.048,Z 334.643,A -85,B 0,C 180,E1 -12521.864,E2 -12521.864} C_VEL
LIN {X 0,Y 376.056,Z 334.639,A -85,B 0,C 180,E1 -12525.168,E2 -12525.168} C_VEL
LIN {X 0,Y 376.022,Z 334.646,A -85,B 0,C 180,E1 -12528.526,E2 -12528.526} C_VEL
LIN {X 0,Y 375.961,Z 334.655,A -85,B 0,C 180,E1 -12531.955,E2 -12531.955} C_VEL
LIN {X 0,Y 376.004,Z 334.646,A -85,B 0,C 180,E1 -12535.462,E2 -12535.462} C_VEL
LIN {X 0,Y 375.975,Z 334.651,A -85,B 0,C 180,E1 -12538.196,E2 -12538.196} C_VEL
LIN {X 0,Y 375.306,Z 334.734,A -85,B 0,C 180,E1 -12539.09,E2 -12539.09} C_VEL
LIN {X 0,Y 372.422,Z 335.094,A -85,B 0,C 180,E1 -12540.542,E2 -12540.542} C_VEL
LIN {X 0,Y 369.991,Z 335.397,A -85,B 0,C 180,E1 -12541.717,E2 -12541.717} C_VEL
LIN {X 0,Y 368.966,Z 335.524,A -85,B 0,C 180,E1 -12542.626,E2 -12542.626} C_VEL
LIN {X 0,Y 368.893,Z 335.532,A -85,B 0,C 180,E1 -12542.934,E2 -12542.934} C_VEL
LIN {X 0,Y 368.917,Z 335.532,A -85,B 0,C 180,E1 -12546.197,E2 -12546.197} C_VEL
LIN {X 0,Y 368.904,Z 335.53,A -85,B 0,C 180,E1 -12548.954,E2 -12548.954} C_VEL
LIN {X 0,Y 368.881,Z 335.538,A -85,B 0,C 180,E1 -12552.01,E2 -12552.01} C_VEL
LIN {X 0,Y 368.88,Z 335.533,A -85,B 0,C 180,E1 -12555.177,E2 -12555.177} C_VEL
LIN {X 0,Y 368.883,Z 335.536,A -85,B 0,C 180,E1 -12558.178,E2 -12558.178} C_VEL
LIN {X 0,Y 368.907,Z 335.531,A -85,B 0,C 180,E1 -12561.361,E2 -12561.361} C_VEL
LIN {X 0,Y 368.937,Z 335.526,A -85,B 0,C 180,E1 -12565.147,E2 -12565.147} C_VEL
LIN {X 0,Y 368.93,Z 335.527,A -85,B 0,C 180,E1 -12569.047,E2 -12569.047} C_VEL
LIN {X 0,Y 369.014,Z 335.52,A -85,B 0,C 180,E1 -12571.975,E2 -12571.975} C_VEL
LIN {X 0,Y 374.786,Z 352.999,A -85,B 0,C 180,E1 -12572.657,E2 -12572.657} C_VEL
LIN {X 0,Y 373.383,Z 423.318,A -85,B 0,C 180,E1 -12574.348,E2 -12574.348} C_VEL
LIN {X 0,Y 373.195,Z 436.945,A -85,B 0,C 180,E1 -12574.916,E2 -12574.916} C_VEL
LIN {X 0,Y 372.721,Z 450.461,A -85,B 0,C 180,E1 -12575.714,E2 -12575.714} C_VEL
LIN {X 0,Y 372.22,Z 462.208,A -85,B 0,C 180,E1 -12576.641,E2 -12576.641} C_VEL
LIN {X 0,Y 371.649,Z 473.673,A -85,B 0,C 180,E1 -12577.778,E2 -12577.778} C_VEL
LIN {X 0,Y 371.014,Z 483.97,A -85,B 0,C 180,E1 -12579.051,E2 -12579.051} C_VEL
LIN {X 0,Y 370.365,Z 492.427,A -85,B 0,C 180,E1 -12580.317,E2 -12580.317} C_VEL
LIN {X 0,Y 369.794,Z 501.589,A -85,B 0,C 180,E1 -12581.997,E2 -12581.997} C_VEL
LIN {X 0,Y 369.328,Z 508.934,A -85,B 0,C 180,E1 -12583.7,E2 -12583.7} C_VEL
LIN {X 0,Y 368.911,Z 515.58,A -85,B 0,C 180,E1 -12585.662,E2 -12585.662} C_VEL
LIN {X 0,Y 368.738,Z 519.843,A -85,B 0,C 180,E1 -12587.339,E2 -12587.339} C_VEL
LIN {X 0,Y 368.561,Z 522.982,A -85,B 0,C 180,E1 -12589.008,E2 -12589.008} C_VEL
LIN {X 0,Y 368.541,Z 524.495,A -85,B 0,C 180,E1 -12590.118,E2 -12590.118} C_VEL
LIN {X 0,Y 368.605,Z 525.572,A -85,B 0,C 180,E1 -12591.227,E2 -12591.227} C_VEL
LIN {X 0,Y 368.714,Z 526.184,A -85,B 0,C 180,E1 -12592.382,E2 -12592.382} C_VEL
LIN {X 0,Y 368.786,Z 526.362,A -85,B 0,C 180,E1 -12593.435,E2 -12593.435} C_VEL
LIN {X 0,Y 368.862,Z 526.15,A -85,B 0,C 180,E1 -12594.534,E2 -12594.534} C_VEL
LIN {X 0,Y 368.936,Z 525.478,A -85,B 0,C 180,E1 -12595.63,E2 -12595.63} C_VEL
LIN {X 0,Y 369.235,Z 524.366,A -85,B 0,C 180,E1 -12596.727,E2 -12596.727} C_VEL
LIN {X 0,Y 369.709,Z 521.884,A -85,B 0,C 180,E1 -12598.367,E2 -12598.367} C_VEL
LIN {X 0,Y 370.27,Z 518.359,A -85,B 0,C 180,E1 -12600.001,E2 -12600.001} C_VEL
LIN {X 0,Y 371.014,Z 513.676,A -85,B 0,C 180,E1 -12601.629,E2 -12601.629} C_VEL
LIN {X 0,Y 371.978,Z 506.541,A -85,B 0,C 180,E1 -12603.521,E2 -12603.521} C_VEL
LIN {X 0,Y 373.056,Z 498.797,A -85,B 0,C 180,E1 -12605.134,E2 -12605.134} C_VEL
LIN {X 0,Y 373.979,Z 490.865,A -85,B 0,C 180,E1 -12606.475,E2 -12606.475} C_VEL
LIN {X 0,Y 375.049,Z 481.129,A -85,B 0,C 180,E1 -12607.809,E2 -12607.809} C_VEL
LIN {X 0,Y 375.969,Z 470.351,A -85,B 0,C 180,E1 -12609.007,E2 -12609.007} C_VEL
LIN {X 0,Y 376.928,Z 458.02,A -85,B 0,C 180,E1 -12610.068,E2 -12610.068} C_VEL
LIN {X 0,Y 377.547,Z 446.054,A -85,B 0,C 180,E1 -12610.864,E2 -12610.864} C_VEL
LIN {X 0,Y 378.014,Z 432.335,A -85,B 0,C 180,E1 -12611.529,E2 -12611.529} C_VEL
LIN {X 0,Y 378.354,Z 414.225,A -85,B 0,C 180,E1 -12612.083,E2 -12612.083} C_VEL
LIN {X 0,Y 380.547,Z 358.77,A -85,B 0,C 180,E1 -12613.557,E2 -12613.557} C_VEL
LIN {X 0,Y 375.385,Z 347.837,A -85,B 0,C 180,E1 -12614.417,E2 -12614.417} C_VEL
LIN {X 0,Y 370.43,Z 338.943,A -85,B 0,C 180,E1 -12615.238,E2 -12615.238} C_VEL
LIN {X 0,Y 369.151,Z 336.32,A -85,B 0,C 180,E1 -12615.476,E2 -12615.476} C_VEL
LIN {X 0,Y 368.985,Z 335.526,A -85,B 0,C 180,E1 -12615.537,E2 -12615.537} C_VEL
LIN {X 0,Y 368.916,Z 335.534,A -85,B 0,C 180,E1 -12618.897,E2 -12618.897} C_VEL
LIN {X 0,Y 368.898,Z 335.535,A -85,B 0,C 180,E1 -12622.398,E2 -12622.398} C_VEL
LIN {X 0,Y 368.923,Z 335.533,A -85,B 0,C 180,E1 -12625.987,E2 -12625.987} C_VEL
LIN {X 0,Y 368.897,Z 335.535,A -85,B 0,C 180,E1 -12629.692,E2 -12629.692} C_VEL
LIN {X 0,Y 368.9,Z 335.531,A -85,B 0,C 180,E1 -12633.043,E2 -12633.043} C_VEL
LIN {X 0,Y 368.914,Z 335.528,A -85,B 0,C 180,E1 -12636.198,E2 -12636.198} C_VEL
LIN {X 0,Y 368.877,Z 335.532,A -85,B 0,C 180,E1 -12638.957,E2 -12638.957} C_VEL
LIN {X 0,Y 368.868,Z 335.536,A -85,B 0,C 180,E1 -12642.006,E2 -12642.006} C_VEL
LIN {X 0,Y 368.88,Z 335.535,A -85,B 0,C 180,E1 -12645.175,E2 -12645.175} C_VEL
LIN {X 0,Y 368.873,Z 335.537,A -85,B 0,C 180,E1 -12648.176,E2 -12648.176} C_VEL
LIN {X 0,Y 368.88,Z 335.537,A -85,B 0,C 180,E1 -12651.366,E2 -12651.366} C_VEL
LIN {X 0,Y 368.94,Z 335.53,A -85,B 0,C 180,E1 -12655.146,E2 -12655.146} C_VEL
LIN {X 0,Y 368.977,Z 335.592,A -85,B 0,C 180,E1 -12656.793,E2 -12656.793} C_VEL
LIN {X 0,Y 372.846,Z 353.41,A -85,B 0,C 180,E1 -12660.356,E2 -12660.356} C_VEL
LIN {X 0,Y 373.841,Z 358.585,A -85,B 0,C 180,E1 -12661.354,E2 -12661.354} C_VEL
LIN {X 0,Y 373.423,Z 365.347,A -85,B 0,C 180,E1 -12662.574,E2 -12662.574} C_VEL
LIN {X 0,Y 371.527,Z 387.776,A -85,B 0,C 180,E1 -12666.557,E2 -12666.557} C_VEL
LIN {X 0,Y 375.169,Z 414.029,A -85,B 0,C 180,E1 -12667.752,E2 -12667.752} C_VEL
LIN {X 0,Y 376.912,Z 432.092,A -85,B 0,C 180,E1 -12668.462,E2 -12668.462} C_VEL
LIN {X 0,Y 377.824,Z 446.644,A -85,B 0,C 180,E1 -12668.981,E2 -12668.981} C_VEL
LIN {X 0,Y 375.806,Z 508.248,A -85,B 0,C 180,E1 -12670.613,E2 -12670.613} C_VEL
LIN {X 0,Y 374.872,Z 521.139,A -85,B 0,C 180,E1 -12671.131,E2 -12671.131} C_VEL
LIN {X 0,Y 373.841,Z 532.874,A -85,B 0,C 180,E1 -12671.787,E2 -12671.787} C_VEL
LIN {X 0,Y 372.625,Z 545.472,A -85,B 0,C 180,E1 -12672.719,E2 -12672.719} C_VEL
LIN {X 0,Y 371.448,Z 556.962,A -85,B 0,C 180,E1 -12673.795,E2 -12673.795} C_VEL
LIN {X 0,Y 370.283,Z 567.422,A -85,B 0,C 180,E1 -12675.012,E2 -12675.012} C_VEL
LIN {X 0,Y 369.439,Z 576.916,A -85,B 0,C 180,E1 -12676.373,E2 -12676.373} C_VEL
LIN {X 0,Y 368.687,Z 585.667,A -85,B 0,C 180,E1 -12677.896,E2 -12677.896} C_VEL
LIN {X 0,Y 368.173,Z 593.439,A -85,B 0,C 180,E1 -12679.552,E2 -12679.552} C_VEL
LIN {X 0,Y 367.976,Z 599.692,A -85,B 0,C 180,E1 -12681.211,E2 -12681.211} C_VEL
LIN {X 0,Y 367.949,Z 604.796,A -85,B 0,C 180,E1 -12682.923,E2 -12682.923} C_VEL
LIN {X 0,Y 368.051,Z 608.446,A -85,B 0,C 180,E1 -12684.521,E2 -12684.521} C_VEL
LIN {X 0,Y 368.239,Z 612.353,A -85,B 0,C 180,E1 -12686.717,E2 -12686.717} C_VEL
LIN {X 0,Y 368.228,Z 613.685,A -85,B 0,C 180,E1 -12687.812,E2 -12687.812} C_VEL
LIN {X 0,Y 368.243,Z 614.566,A -85,B 0,C 180,E1 -12688.906,E2 -12688.906} C_VEL
LIN {X 0,Y 368.277,Z 615.007,A -85,B 0,C 180,E1 -12690,E2 -12690} C_VEL
LIN {X 0,Y 368.193,Z 614.956,A -85,B 0,C 180,E1 -12691.094,E2 -12691.094} C_VEL
LIN {X 0,Y 368.149,Z 614.438,A -85,B 0,C 180,E1 -12692.188,E2 -12692.188} C_VEL
LIN {X 0,Y 368.22,Z 613.501,A -85,B 0,C 180,E1 -12693.282,E2 -12693.282} C_VEL
LIN {X 0,Y 368.084,Z 612.097,A -85,B 0,C 180,E1 -12694.38,E2 -12694.38} C_VEL
LIN {X 0,Y 367.911,Z 608.515,A -85,B 0,C 180,E1 -12696.286,E2 -12696.286} C_VEL
LIN {X 0,Y 367.878,Z 603.352,A -85,B 0,C 180,E1 -12698.238,E2 -12698.238} C_VEL
LIN {X 0,Y 368.044,Z 597.67,A -85,B 0,C 180,E1 -12699.896,E2 -12699.896} C_VEL
LIN {X 0,Y 368.487,Z 590.635,A -85,B 0,C 180,E1 -12701.552,E2 -12701.552} C_VEL
LIN {X 0,Y 369.252,Z 581.956,A -85,B 0,C 180,E1 -12703.203,E2 -12703.203} C_VEL
LIN {X 0,Y 370.041,Z 573.198,A -85,B 0,C 180,E1 -12704.575,E2 -12704.575} C_VEL
LIN {X 0,Y 371.18,Z 562.706,A -85,B 0,C 180,E1 -12705.935,E2 -12705.935} C_VEL
LIN {X 0,Y 372.571,Z 551.085,A -85,B 0,C 180,E1 -12707.142,E2 -12707.142} C_VEL
LIN {X 0,Y 373.999,Z 538.224,A -85,B 0,C 180,E1 -12708.204,E2 -12708.204} C_VEL
LIN {X 0,Y 375.252,Z 525.861,A -85,B 0,C 180,E1 -12708.99,E2 -12708.99} C_VEL
LIN {X 0,Y 376.471,Z 511.203,A -85,B 0,C 180,E1 -12709.67,E2 -12709.67} C_VEL
LIN {X 0,Y 377.124,Z 496.611,A -85,B 0,C 180,E1 -12710.132,E2 -12710.132} C_VEL
LIN {X 0,Y 379.096,Z 444.423,A -85,B 0,C 180,E1 -12711.56,E2 -12711.56} C_VEL
LIN {X 0,Y 377.751,Z 424.612,A -85,B 0,C 180,E1 -12712.324,E2 -12712.324} C_VEL
LIN {X 0,Y 375.74,Z 408.533,A -85,B 0,C 180,E1 -12713.06,E2 -12713.06} C_VEL
LIN {X 0,Y 372.622,Z 390.85,A -85,B 0,C 180,E1 -12714.033,E2 -12714.033} C_VEL
LIN {X 0,Y 374.702,Z 374.04,A -85,B 0,C 180,E1 -12717.357,E2 -12717.357} C_VEL
LIN {X 0,Y 376.087,Z 364.253,A -85,B 0,C 180,E1 -12719.376,E2 -12719.376} C_VEL
LIN {X 0,Y 374.701,Z 356.414,A -85,B 0,C 180,E1 -12721.365,E2 -12721.365} C_VEL
LIN {X 0,Y 372.549,Z 347.639,A -85,B 0,C 180,E1 -12723.896,E2 -12723.896} C_VEL
LIN {X 0,Y 370.681,Z 341.279,A -85,B 0,C 180,E1 -12725.998,E2 -12725.998} C_VEL
LIN {X 0,Y 368.897,Z 335.536,A -85,B 0,C 180,E1 -12728.256,E2 -12728.256} C_VEL
LIN {X 0,Y 368.873,Z 335.54,A -85,B 0,C 180,E1 -12732.007,E2 -12732.007} C_VEL
LIN {X 0,Y 368.881,Z 335.537,A -85,B 0,C 180,E1 -12735.175,E2 -12735.175} C_VEL
LIN {X 0,Y 368.871,Z 335.538,A -85,B 0,C 180,E1 -12738.175,E2 -12738.175} C_VEL
LIN {X 0,Y 368.878,Z 335.536,A -85,B 0,C 180,E1 -12741.366,E2 -12741.366} C_VEL
LIN {X 0,Y 368.932,Z 335.529,A -85,B 0,C 180,E1 -12745.145,E2 -12745.145} C_VEL
LIN {X 0,Y 368.915,Z 335.533,A -85,B 0,C 180,E1 -12749.045,E2 -12749.045} C_VEL
LIN {X 0,Y 368.909,Z 335.534,A -85,B 0,C 180,E1 -12751.557,E2 -12751.557} C_VEL
LIN {X 0,Y 368.887,Z 335.538,A -85,B 0,C 180,E1 -12755.219,E2 -12755.219} C_VEL
LIN {X 0,Y 368.944,Z 335.667,A -85,B 0,C 180,E1 -12757.884,E2 -12757.884} C_VEL
LIN {X 0,Y 369.97,Z 338.472,A -85,B 0,C 180,E1 -12758.132,E2 -12758.132} C_VEL
LIN {X 0,Y 371.495,Z 340.716,A -85,B 0,C 180,E1 -12758.411,E2 -12758.411} C_VEL
LIN {X 0,Y 376.949,Z 350.398,A -85,B 0,C 180,E1 -12759.422,E2 -12759.422} C_VEL
LIN {X 0,Y 381.642,Z 360.03,A -85,B 0,C 180,E1 -12760.269,E2 -12760.269} C_VEL
LIN {X 0,Y 378.781,Z 422.065,A -85,B 0,C 180,E1 -12762.033,E2 -12762.033} C_VEL
LIN {X 0,Y 378.523,Z 436.23,A -85,B 0,C 180,E1 -12762.544,E2 -12762.544} C_VEL
LIN {X 0,Y 377.973,Z 449.532,A -85,B 0,C 180,E1 -12763.249,E2 -12763.249} C_VEL
LIN {X 0,Y 377.28,Z 460.891,A -85,B 0,C 180,E1 -12764.052,E2 -12764.052} C_VEL
LIN {X 0,Y 376.282,Z 472.653,A -85,B 0,C 180,E1 -12765.118,E2 -12765.118} C_VEL
LIN {X 0,Y 375.265,Z 483.23,A -85,B 0,C 180,E1 -12766.323,E2 -12766.323} C_VEL
LIN {X 0,Y 374.317,Z 491.699,A -85,B 0,C 180,E1 -12767.509,E2 -12767.509} C_VEL
LIN {X 0,Y 373.098,Z 501.144,A -85,B 0,C 180,E1 -12769.142,E2 -12769.142} C_VEL
LIN {X 0,Y 372.027,Z 508.607,A -85,B 0,C 180,E1 -12770.759,E2 -12770.759} C_VEL
LIN {X 0,Y 371.17,Z 514.489,A -85,B 0,C 180,E1 -12772.383,E2 -12772.383} C_VEL
LIN {X 0,Y 370.388,Z 519.123,A -85,B 0,C 180,E1 -12774.009,E2 -12774.009} C_VEL
LIN {X 0,Y 369.761,Z 522.607,A -85,B 0,C 180,E1 -12775.639,E2 -12775.639} C_VEL
LIN {X 0,Y 369.431,Z 524.347,A -85,B 0,C 180,E1 -12776.728,E2 -12776.728} C_VEL
LIN {X 0,Y 369.247,Z 525.621,A -85,B 0,C 180,E1 -12777.818,E2 -12777.818} C_VEL
LIN {X 0,Y 369.055,Z 526.447,A -85,B 0,C 180,E1 -12778.908,E2 -12778.908} C_VEL
LIN {X 0,Y 368.933,Z 526.862,A -85,B 0,C 180,E1 -12779.999,E2 -12779.999} C_VEL
LIN {X 0,Y 368.736,Z 526.883,A -85,B 0,C 180,E1 -12781.092,E2 -12781.092} C_VEL
LIN {X 0,Y 368.409,Z 526.455,A -85,B 0,C 180,E1 -12782.186,E2 -12782.186} C_VEL
LIN {X 0,Y 368.428,Z 525.576,A -85,B 0,C 180,E1 -12783.28,E2 -12783.28} C_VEL
LIN {X 0,Y 368.621,Z 524.276,A -85,B 0,C 180,E1 -12784.373,E2 -12784.373} C_VEL
LIN {X 0,Y 368.784,Z 521.487,A -85,B 0,C 180,E1 -12786.016,E2 -12786.016} C_VEL
LIN {X 0,Y 368.849,Z 517.349,A -85,B 0,C 180,E1 -12787.776,E2 -12787.776} C_VEL
LIN {X 0,Y 369.119,Z 512.625,A -85,B 0,C 180,E1 -12789.313,E2 -12789.313} C_VEL
LIN {X 0,Y 369.486,Z 506.252,A -85,B 0,C 180,E1 -12790.964,E2 -12790.964} C_VEL
LIN {X 0,Y 369.981,Z 498.323,A -85,B 0,C 180,E1 -12792.617,E2 -12792.617} C_VEL
LIN {X 0,Y 370.486,Z 490.237,A -85,B 0,C 180,E1 -12793.996,E2 -12793.996} C_VEL
LIN {X 0,Y 371.019,Z 480.353,A -85,B 0,C 180,E1 -12795.378,E2 -12795.378} C_VEL
LIN {X 0,Y 371.693,Z 469.399,A -85,B 0,C 180,E1 -12796.617,E2 -12796.617} C_VEL
LIN {X 0,Y 372.171,Z 458.876,A -85,B 0,C 180,E1 -12797.586,E2 -12797.586} C_VEL
LIN {X 0,Y 372.765,Z 446.48,A -85,B 0,C 180,E1 -12798.48,E2 -12798.48} C_VEL
LIN {X 0,Y 373.141,Z 432.322,A -85,B 0,C 180,E1 -12799.242,E2 -12799.242} C_VEL
LIN {X 0,Y 373.271,Z 418.647,A -85,B 0,C 180,E1 -12799.731,E2 -12799.731} C_VEL
LIN {X 0,Y 374.591,Z 352.753,A -85,B 0,C 180,E1 -12801.343,E2 -12801.343} C_VEL
LIN {X 0,Y 368.934,Z 335.529,A -85,B 0,C 180,E1 -12802.03,E2 -12802.03} C_VEL
LIN {X 0,Y 368.958,Z 335.528,A -85,B 0,C 180,E1 -12804.775,E2 -12804.775} C_VEL
LIN {X 0,Y 368.968,Z 335.524,A -85,B 0,C 180,E1 -12807.202,E2 -12807.202} C_VEL
LIN {X 0,Y 368.918,Z 335.528,A -85,B 0,C 180,E1 -12809.689,E2 -12809.689} C_VEL
LIN {X 0,Y 368.896,Z 335.534,A -85,B 0,C 180,E1 -12813.043,E2 -12813.043} C_VEL
LIN {X 0,Y 368.916,Z 335.529,A -85,B 0,C 180,E1 -12816.196,E2 -12816.196} C_VEL
LIN {X 0,Y 368.9,Z 335.534,A -85,B 0,C 180,E1 -12818.953,E2 -12818.953} C_VEL
LIN {X 0,Y 368.879,Z 335.533,A -85,B 0,C 180,E1 -12822.009,E2 -12822.009} C_VEL
LIN {X 0,Y 368.882,Z 335.535,A -85,B 0,C 180,E1 -12825.176,E2 -12825.176} C_VEL
LIN {X 0,Y 368.881,Z 335.534,A -85,B 0,C 180,E1 -12828.177,E2 -12828.177} C_VEL
LIN {X 0,Y 368.908,Z 335.53,A -85,B 0,C 180,E1 -12831.359,E2 -12831.359} C_VEL
LIN {X 0,Y 368.934,Z 335.528,A -85,B 0,C 180,E1 -12835.146,E2 -12835.146} C_VEL
LIN {X 0,Y 368.926,Z 335.529,A -85,B 0,C 180,E1 -12839.046,E2 -12839.046} C_VEL
LIN {X 0,Y 368.96,Z 335.526,A -85,B 0,C 180,E1 -12842.796,E2 -12842.796} C_VEL
LIN {X 0,Y 368.942,Z 335.527,A -85,B 0,C 180,E1 -12846.113,E2 -12846.113} C_VEL
LIN {X 0,Y 368.934,Z 335.527,A -85,B 0,C 180,E1 -12849.947,E2 -12849.947} C_VEL
LIN {X 0,Y 368.973,Z 335.522,A -85,B 0,C 180,E1 -12853.399,E2 -12853.399} C_VEL
LIN {X 0,Y 369.055,Z 335.514,A -85,B 0,C 180,E1 -12856.79,E2 -12856.79} C_VEL
LIN {X 0,Y 369.067,Z 335.513,A -85,B 0,C 180,E1 -12860.132,E2 -12860.132} C_VEL
LIN {X 0,Y 369.186,Z 335.5,A -85,B 0,C 180,E1 -12862.342,E2 -12862.342} C_VEL
LIN {X 0,Y 369.142,Z 335.504,A -85,B 0,C 180,E1 -12864.538,E2 -12864.538} C_VEL
LIN {X 0,Y 369.316,Z 335.48,A -85,B 0,C 180,E1 -12867.819,E2 -12867.819} C_VEL
LIN {X 0,Y 369.456,Z 335.464,A -85,B 0,C 180,E1 -12870,E2 -12870} C_VEL
LIN {X 0,Y 369.316,Z 335.483,A -85,B 0,C 180,E1 -12872.181,E2 -12872.181} C_VEL
LIN {X 0,Y 369.206,Z 335.496,A -85,B 0,C 180,E1 -12876.558,E2 -12876.558} C_VEL
LIN {X 0,Y 369.135,Z 335.504,A -85,B 0,C 180,E1 -12878.761,E2 -12878.761} C_VEL
LIN {X 0,Y 369.003,Z 335.522,A -85,B 0,C 180,E1 -12882.094,E2 -12882.094} C_VEL
LIN {X 0,Y 368.996,Z 335.519,A -85,B 0,C 180,E1 -12885.465,E2 -12885.465} C_VEL
LIN {X 0,Y 368.98,Z 335.521,A -85,B 0,C 180,E1 -12888.893,E2 -12888.893} C_VEL
LIN {X 0,Y 368.931,Z 335.53,A -85,B 0,C 180,E1 -12892.396,E2 -12892.396} C_VEL
LIN {X 0,Y 368.998,Z 335.523,A -85,B 0,C 180,E1 -12895.981,E2 -12895.981} C_VEL
LIN {X 0,Y 368.913,Z 335.531,A -85,B 0,C 180,E1 -12899.691,E2 -12899.691} C_VEL
LIN {X 0,Y 368.893,Z 335.532,A -85,B 0,C 180,E1 -12902.934,E2 -12902.934} C_VEL
LIN {X 0,Y 368.251,Z 335.615,A -85,B 0,C 180,E1 -12903.845,E2 -12903.845} C_VEL
LIN {X 0,Y 365.4,Z 335.967,A -85,B 0,C 180,E1 -12905.326,E2 -12905.326} C_VEL
LIN {X 0,Y 362.97,Z 336.272,A -85,B 0,C 180,E1 -12906.524,E2 -12906.524} C_VEL
LIN {X 0,Y 361.929,Z 336.4,A -85,B 0,C 180,E1 -12907.451,E2 -12907.451} C_VEL
LIN {X 0,Y 361.847,Z 336.408,A -85,B 0,C 180,E1 -12907.765,E2 -12907.765} C_VEL
LIN {X 0,Y 361.827,Z 336.412,A -85,B 0,C 180,E1 -12911.331,E2 -12911.331} C_VEL
LIN {X 0,Y 361.817,Z 336.416,A -85,B 0,C 180,E1 -12914.369,E2 -12914.369} C_VEL
LIN {X 0,Y 361.836,Z 336.412,A -85,B 0,C 180,E1 -12917.569,E2 -12917.569} C_VEL
LIN {X 0,Y 361.868,Z 336.407,A -85,B 0,C 180,E1 -12920.974,E2 -12920.974} C_VEL
LIN {X 0,Y 361.875,Z 336.406,A -85,B 0,C 180,E1 -12924.656,E2 -12924.656} C_VEL
LIN {X 0,Y 361.839,Z 336.412,A -85,B 0,C 180,E1 -12928.371,E2 -12928.371} C_VEL
LIN {X 0,Y 361.964,Z 336.399,A -85,B 0,C 180,E1 -12931.696,E2 -12931.696} C_VEL
LIN {X 0,Y 367.937,Z 354.489,A -85,B 0,C 180,E1 -12932.421,E2 -12932.421} C_VEL
LIN {X 0,Y 366.445,Z 423.81,A -85,B 0,C 180,E1 -12934.13,E2 -12934.13} C_VEL
LIN {X 0,Y 366.299,Z 436.401,A -85,B 0,C 180,E1 -12934.651,E2 -12934.651} C_VEL
LIN {X 0,Y 365.82,Z 450.057,A -85,B 0,C 180,E1 -12935.453,E2 -12935.453} C_VEL
LIN {X 0,Y 365.322,Z 461.322,A -85,B 0,C 180,E1 -12936.323,E2 -12936.323} C_VEL
LIN {X 0,Y 364.699,Z 472.967,A -85,B 0,C 180,E1 -12937.468,E2 -12937.468} C_VEL
LIN {X 0,Y 364.076,Z 483.73,A -85,B 0,C 180,E1 -12938.781,E2 -12938.781} C_VEL
LIN {X 0,Y 363.358,Z 493.237,A -85,B 0,C 180,E1 -12940.216,E2 -12940.216} C_VEL
LIN {X 0,Y 362.744,Z 502.492,A -85,B 0,C 180,E1 -12941.942,E2 -12941.942} C_VEL
LIN {X 0,Y 362.275,Z 509.798,A -85,B 0,C 180,E1 -12943.663,E2 -12943.663} C_VEL
LIN {X 0,Y 361.899,Z 515.613,A -85,B 0,C 180,E1 -12945.378,E2 -12945.378} C_VEL
LIN {X 0,Y 361.715,Z 520.119,A -85,B 0,C 180,E1 -12947.089,E2 -12947.089} C_VEL
LIN {X 0,Y 361.519,Z 523.456,A -85,B 0,C 180,E1 -12948.791,E2 -12948.791} C_VEL
LIN {X 0,Y 361.511,Z 525.062,A -85,B 0,C 180,E1 -12949.924,E2 -12949.924} C_VEL
LIN {X 0,Y 361.541,Z 526.242,A -85,B 0,C 180,E1 -12951.054,E2 -12951.054} C_VEL
LIN {X 0,Y 361.68,Z 527.042,A -85,B 0,C 180,E1 -12952.315,E2 -12952.315} C_VEL
LIN {X 0,Y 361.837,Z 527.167,A -85,B 0,C 180,E1 -12954.427,E2 -12954.427} C_VEL
LIN {X 0,Y 361.911,Z 526.65,A -85,B 0,C 180,E1 -12955.546,E2 -12955.546} C_VEL
LIN {X 0,Y 362.219,Z 525.628,A -85,B 0,C 180,E1 -12956.664,E2 -12956.664} C_VEL
LIN {X 0,Y 362.529,Z 524.199,A -85,B 0,C 180,E1 -12957.778,E2 -12957.778} C_VEL
LIN {X 0,Y 363.084,Z 521.201,A -85,B 0,C 180,E1 -12959.446,E2 -12959.446} C_VEL
LIN {X 0,Y 363.798,Z 517.111,A -85,B 0,C 180,E1 -12961.107,E2 -12961.107} C_VEL
LIN {X 0,Y 364.804,Z 510.796,A -85,B 0,C 180,E1 -12963.037,E2 -12963.037} C_VEL
LIN {X 0,Y 365.815,Z 503.876,A -85,B 0,C 180,E1 -12964.684,E2 -12964.684} C_VEL
LIN {X 0,Y 366.786,Z 496.792,A -85,B 0,C 180,E1 -12966.05,E2 -12966.05} C_VEL
LIN {X 0,Y 367.8,Z 488.214,A -85,B 0,C 180,E1 -12967.411,E2 -12967.411} C_VEL
LIN {X 0,Y 368.983,Z 477.553,A -85,B 0,C 180,E1 -12968.765,E2 -12968.765} C_VEL
LIN {X 0,Y 369.923,Z 467.115,A -85,B 0,C 180,E1 -12969.846,E2 -12969.846} C_VEL
LIN {X 0,Y 370.857,Z 455.438,A -85,B 0,C 180,E1 -12970.786,E2 -12970.786} C_VEL
LIN {X 0,Y 371.465,Z 442.458,A -85,B 0,C 180,E1 -12971.597,E2 -12971.597} C_VEL
LIN {X 0,Y 371.841,Z 429.173,A -85,B 0,C 180,E1 -12972.173,E2 -12972.173} C_VEL
LIN {X 0,Y 372.765,Z 398.317,A -85,B 0,C 180,E1 -12973.042,E2 -12973.042} C_VEL
LIN {X 0,Y 374.443,Z 360.956,A -85,B 0,C 180,E1 -12974.078,E2 -12974.078} C_VEL
LIN {X 0,Y 369.994,Z 351.571,A -85,B 0,C 180,E1 -12974.852,E2 -12974.852} C_VEL
LIN {X 0,Y 363.743,Z 340.29,A -85,B 0,C 180,E1 -12975.968,E2 -12975.968} C_VEL
LIN {X 0,Y 362.187,Z 337.601,A -85,B 0,C 180,E1 -12976.256,E2 -12976.256} C_VEL
LIN {X 0,Y 361.935,Z 336.401,A -85,B 0,C 180,E1 -12976.353,E2 -12976.353} C_VEL
LIN {X 0,Y 361.854,Z 336.417,A -85,B 0,C 180,E1 -12979.28,E2 -12979.28} C_VEL
LIN {X 0,Y 361.864,Z 336.408,A -85,B 0,C 180,E1 -12982.858,E2 -12982.858} C_VEL
LIN {X 0,Y 361.858,Z 336.413,A -85,B 0,C 180,E1 -12986.533,E2 -12986.533} C_VEL
LIN {X 0,Y 361.859,Z 336.411,A -85,B 0,C 180,E1 -12990.33,E2 -12990.33} C_VEL
LIN {X 0,Y 361.854,Z 336.41,A -85,B 0,C 180,E1 -12994.281,E2 -12994.281} C_VEL
LIN {X 0,Y 361.861,Z 336.406,A -85,B 0,C 180,E1 -12997.221,E2 -12997.221} C_VEL
LIN {X 0,Y 361.814,Z 336.411,A -85,B 0,C 180,E1 -13000.751,E2 -13000.751} C_VEL
LIN {X 0,Y 361.816,Z 336.414,A -85,B 0,C 180,E1 -13004.369,E2 -13004.369} C_VEL
LIN {X 0,Y 361.834,Z 336.414,A -85,B 0,C 180,E1 -13007.569,E2 -13007.569} C_VEL
LIN {X 0,Y 361.847,Z 336.413,A -85,B 0,C 180,E1 -13011.572,E2 -13011.572} C_VEL
LIN {X 0,Y 361.878,Z 336.408,A -85,B 0,C 180,E1 -13014.655,E2 -13014.655} C_VEL
LIN {X 0,Y 361.97,Z 336.568,A -85,B 0,C 180,E1 -13016.568,E2 -13016.568} C_VEL
LIN {X 0,Y 365.983,Z 355.238,A -85,B 0,C 180,E1 -13020.364,E2 -13020.364} C_VEL
LIN {X 0,Y 366.896,Z 360.462,A -85,B 0,C 180,E1 -13021.387,E2 -13021.387} C_VEL
LIN {X 0,Y 365.29,Z 378.802,A -85,B 0,C 180,E1 -13024.724,E2 -13024.724} C_VEL
LIN {X 0,Y 364.831,Z 384.587,A -85,B 0,C 180,E1 -13025.76,E2 -13025.76} C_VEL
LIN {X 0,Y 368.741,Z 412.778,A -85,B 0,C 180,E1 -13027.113,E2 -13027.113} C_VEL
LIN {X 0,Y 370.537,Z 430.891,A -85,B 0,C 180,E1 -13027.873,E2 -13027.873} C_VEL
LIN {X 0,Y 371.565,Z 448.083,A -85,B 0,C 180,E1 -13028.497,E2 -13028.497} C_VEL
LIN {X 0,Y 369.343,Z 508.041,A -85,B 0,C 180,E1 -13030.151,E2 -13030.151} C_VEL
LIN {X 0,Y 368.335,Z 521.327,A -85,B 0,C 180,E1 -13030.711,E2 -13030.711} C_VEL
LIN {X 0,Y 367.153,Z 533.674,A -85,B 0,C 180,E1 -13031.444,E2 -13031.444} C_VEL
LIN {X 0,Y 365.875,Z 545.872,A -85,B 0,C 180,E1 -13032.39,E2 -13032.39} C_VEL
LIN {X 0,Y 364.646,Z 556.996,A -85,B 0,C 180,E1 -13033.484,E2 -13033.484} C_VEL
LIN {X 0,Y 363.392,Z 567.22,A -85,B 0,C 180,E1 -13034.721,E2 -13034.721} C_VEL
LIN {X 0,Y 362.458,Z 577.006,A -85,B 0,C 180,E1 -13036.171,E2 -13036.171} C_VEL
LIN {X 0,Y 361.701,Z 585.265,A -85,B 0,C 180,E1 -13037.658,E2 -13037.658} C_VEL
LIN {X 0,Y 361.121,Z 592.877,A -85,B 0,C 180,E1 -13039.345,E2 -13039.345} C_VEL
LIN {X 0,Y 360.887,Z 599.047,A -85,B 0,C 180,E1 -13041.037,E2 -13041.037} C_VEL
LIN {X 0,Y 360.857,Z 603.955,A -85,B 0,C 180,E1 -13042.727,E2 -13042.727} C_VEL
LIN {X 0,Y 360.979,Z 607.697,A -85,B 0,C 180,E1 -13044.413,E2 -13044.413} C_VEL
LIN {X 0,Y 361.196,Z 611.248,A -85,B 0,C 180,E1 -13046.653,E2 -13046.653} C_VEL
LIN {X 0,Y 361.191,Z 612.65,A -85,B 0,C 180,E1 -13047.77,E2 -13047.77} C_VEL
LIN {X 0,Y 361.208,Z 613.563,A -85,B 0,C 180,E1 -13048.885,E2 -13048.885} C_VEL
LIN {X 0,Y 361.243,Z 614.037,A -85,B 0,C 180,E1 -13050,E2 -13050} C_VEL
LIN {X 0,Y 361.147,Z 614.046,A -85,B 0,C 180,E1 -13051.115,E2 -13051.115} C_VEL
LIN {X 0,Y 361.1,Z 613.566,A -85,B 0,C 180,E1 -13052.231,E2 -13052.231} C_VEL
LIN {X 0,Y 361.153,Z 612.653,A -85,B 0,C 180,E1 -13053.347,E2 -13053.347} C_VEL
LIN {X 0,Y 360.992,Z 611.28,A -85,B 0,C 180,E1 -13054.466,E2 -13054.466} C_VEL
LIN {X 0,Y 360.825,Z 608.109,A -85,B 0,C 180,E1 -13056.263,E2 -13056.263} C_VEL
LIN {X 0,Y 360.782,Z 604.302,A -85,B 0,C 180,E1 -13057.837,E2 -13057.837} C_VEL
LIN {X 0,Y 360.924,Z 598.124,A -85,B 0,C 180,E1 -13059.81,E2 -13059.81} C_VEL
LIN {X 0,Y 361.37,Z 591.406,A -85,B 0,C 180,E1 -13061.498,E2 -13061.498} C_VEL
LIN {X 0,Y 362.109,Z 583.173,A -85,B 0,C 180,E1 -13063.182,E2 -13063.182} C_VEL
LIN {X 0,Y 362.934,Z 574.888,A -85,B 0,C 180,E1 -13064.58,E2 -13064.58} C_VEL
LIN {X 0,Y 364.213,Z 563.85,A -85,B 0,C 180,E1 -13066.104,E2 -13066.104} C_VEL
LIN {X 0,Y 365.816,Z 551.455,A -85,B 0,C 180,E1 -13067.469,E2 -13067.469} C_VEL
LIN {X 0,Y 367.303,Z 538.964,A -85,B 0,C 180,E1 -13068.548,E2 -13068.548} C_VEL
LIN {X 0,Y 368.722,Z 526.135,A -85,B 0,C 180,E1 -13069.412,E2 -13069.412} C_VEL
LIN {X 0,Y 369.986,Z 512.158,A -85,B 0,C 180,E1 -13070.102,E2 -13070.102} C_VEL
LIN {X 0,Y 370.771,Z 497.781,A -85,B 0,C 180,E1 -13070.601,E2 -13070.601} C_VEL
LIN {X 0,Y 372.986,Z 445.862,A -85,B 0,C 180,E1 -13072.061,E2 -13072.061} C_VEL
LIN {X 0,Y 371.791,Z 426.581,A -85,B 0,C 180,E1 -13072.83,E2 -13072.83} C_VEL
LIN {X 0,Y 369.977,Z 411.043,A -85,B 0,C 180,E1 -13073.566,E2 -13073.566} C_VEL
LIN {X 0,Y 366.623,Z 392.23,A -85,B 0,C 180,E1 -13074.637,E2 -13074.637} C_VEL
LIN {X 0,Y 366.148,Z 389.444,A -85,B 0,C 180,E1 -13074.812,E2 -13074.812} C_VEL
LIN {X 0,Y 368.902,Z 370.047,A -85,B 0,C 180,E1 -13078.794,E2 -13078.794} C_VEL
LIN {X 0,Y 369.421,Z 366.146,A -85,B 0,C 180,E1 -13079.646,E2 -13079.646} C_VEL
LIN {X 0,Y 368.036,Z 358.428,A -85,B 0,C 180,E1 -13081.678,E2 -13081.678} C_VEL
LIN {X 0,Y 365.888,Z 349.634,A -85,B 0,C 180,E1 -13084.315,E2 -13084.315} C_VEL
LIN {X 0,Y 363.797,Z 342.636,A -85,B 0,C 180,E1 -13086.789,E2 -13086.789} C_VEL
LIN {X 0,Y 361.824,Z 336.419,A -85,B 0,C 180,E1 -13089.395,E2 -13089.395} C_VEL
LIN {X 0,Y 361.835,Z 336.415,A -85,B 0,C 180,E1 -13092.829,E2 -13092.829} C_VEL
LIN {X 0,Y 361.819,Z 336.416,A -85,B 0,C 180,E1 -13095.947,E2 -13095.947} C_VEL
LIN {X 0,Y 361.814,Z 336.416,A -85,B 0,C 180,E1 -13099.249,E2 -13099.249} C_VEL
LIN {X 0,Y 361.863,Z 336.408,A -85,B 0,C 180,E1 -13102.981,E2 -13102.981} C_VEL
LIN {X 0,Y 361.86,Z 336.409,A -85,B 0,C 180,E1 -13106.631,E2 -13106.631} C_VEL
LIN {X 0,Y 361.857,Z 336.412,A -85,B 0,C 180,E1 -13109.67,E2 -13109.67} C_VEL
LIN {X 0,Y 361.856,Z 336.414,A -85,B 0,C 180,E1 -13113.467,E2 -13113.467} C_VEL
LIN {X 0,Y 361.863,Z 336.413,A -85,B 0,C 180,E1 -13116.935,E2 -13116.935} C_VEL
LIN {X 0,Y 362.893,Z 339.284,A -85,B 0,C 180,E1 -13117.211,E2 -13117.211} C_VEL
LIN {X 0,Y 364.479,Z 341.435,A -85,B 0,C 180,E1 -13117.526,E2 -13117.526} C_VEL
LIN {X 0,Y 370.86,Z 352.578,A -85,B 0,C 180,E1 -13118.796,E2 -13118.796} C_VEL
LIN {X 0,Y 375.668,Z 362.361,A -85,B 0,C 180,E1 -13119.719,E2 -13119.719} C_VEL
LIN {X 0,Y 372.648,Z 423.255,A -85,B 0,C 180,E1 -13121.513,E2 -13121.513} C_VEL
LIN {X 0,Y 372.355,Z 437.224,A -85,B 0,C 180,E1 -13122.032,E2 -13122.032} C_VEL
LIN {X 0,Y 371.763,Z 450.432,A -85,B 0,C 180,E1 -13122.748,E2 -13122.748} C_VEL
LIN {X 0,Y 370.935,Z 462.598,A -85,B 0,C 180,E1 -13123.63,E2 -13123.63} C_VEL
LIN {X 0,Y 369.885,Z 474.187,A -85,B 0,C 180,E1 -13124.714,E2 -13124.714} C_VEL
LIN {X 0,Y 368.786,Z 484.642,A -85,B 0,C 180,E1 -13125.937,E2 -13125.937} C_VEL
LIN {X 0,Y 367.65,Z 493.869,A -85,B 0,C 180,E1 -13127.279,E2 -13127.279} C_VEL
LIN {X 0,Y 366.388,Z 503.101,A -85,B 0,C 180,E1 -13128.941,E2 -13128.941} C_VEL
LIN {X 0,Y 365.223,Z 510.331,A -85,B 0,C 180,E1 -13130.586,E2 -13130.586} C_VEL
LIN {X 0,Y 364.3,Z 516.072,A -85,B 0,C 180,E1 -13132.238,E2 -13132.238} C_VEL
LIN {X 0,Y 363.491,Z 520.567,A -85,B 0,C 180,E1 -13133.895,E2 -13133.895} C_VEL
LIN {X 0,Y 362.825,Z 523.921,A -85,B 0,C 180,E1 -13135.556,E2 -13135.556} C_VEL
LIN {X 0,Y 362.473,Z 525.591,A -85,B 0,C 180,E1 -13136.665,E2 -13136.665} C_VEL
LIN {X 0,Y 362.245,Z 526.765,A -85,B 0,C 180,E1 -13137.776,E2 -13137.776} C_VEL
LIN {X 0,Y 362.039,Z 527.526,A -85,B 0,C 180,E1 -13138.887,E2 -13138.887} C_VEL
LIN {X 0,Y 361.915,Z 527.876,A -85,B 0,C 180,E1 -13139.999,E2 -13139.999} C_VEL
LIN {X 0,Y 361.701,Z 527.792,A -85,B 0,C 180,E1 -13141.113,E2 -13141.113} C_VEL
LIN {X 0,Y 361.361,Z 527.291,A -85,B 0,C 180,E1 -13142.229,E2 -13142.229} C_VEL
LIN {X 0,Y 361.387,Z 526.346,A -85,B 0,C 180,E1 -13143.344,E2 -13143.344} C_VEL
LIN {X 0,Y 361.593,Z 524.953,A -85,B 0,C 180,E1 -13144.458,E2 -13144.458} C_VEL
LIN {X 0,Y 361.744,Z 522.035,A -85,B 0,C 180,E1 -13146.133,E2 -13146.133} C_VEL
LIN {X 0,Y 361.789,Z 518.049,A -85,B 0,C 180,E1 -13147.815,E2 -13147.815} C_VEL
LIN {X 0,Y 362.091,Z 512.857,A -85,B 0,C 180,E1 -13149.496,E2 -13149.496} C_VEL
LIN {X 0,Y 362.467,Z 506.318,A -85,B 0,C 180,E1 -13151.18,E2 -13151.18} C_VEL
LIN {X 0,Y 362.985,Z 498.192,A -85,B 0,C 180,E1 -13152.865,E2 -13152.865} C_VEL
LIN {X 0,Y 363.514,Z 489.838,A -85,B 0,C 180,E1 -13154.27,E2 -13154.27} C_VEL
LIN {X 0,Y 364.106,Z 479.645,A -85,B 0,C 180,E1 -13155.677,E2 -13155.677} C_VEL
LIN {X 0,Y 364.717,Z 469.702,A -85,B 0,C 180,E1 -13156.8,E2 -13156.8} C_VEL
LIN {X 0,Y 365.195,Z 459.041,A -85,B 0,C 180,E1 -13157.788,E2 -13157.788} C_VEL
LIN {X 0,Y 365.786,Z 446.418,A -85,B 0,C 180,E1 -13158.7,E2 -13158.7} C_VEL
LIN {X 0,Y 366.163,Z 433.083,A -85,B 0,C 180,E1 -13159.425,E2 -13159.425} C_VEL
LIN {X 0,Y 366.313,Z 419.212,A -85,B 0,C 180,E1 -13159.93,E2 -13159.93} C_VEL
LIN {X 0,Y 367.695,Z 354.178,A -85,B 0,C 180,E1 -13161.571,E2 -13161.571} C_VEL
LIN {X 0,Y 361.893,Z 336.407,A -85,B 0,C 180,E1 -13162.279,E2 -13162.279} C_VEL
LIN {X 0,Y 361.928,Z 336.401,A -85,B 0,C 180,E1 -13165.289,E2 -13165.289} C_VEL
LIN {X 0,Y 361.918,Z 336.4,A -85,B 0,C 180,E1 -13167.778,E2 -13167.778} C_VEL
LIN {X 0,Y 361.846,Z 336.411,A -85,B 0,C 180,E1 -13171.285,E2 -13171.285} C_VEL
LIN {X 0,Y 361.853,Z 336.409,A -85,B 0,C 180,E1 -13174.28,E2 -13174.28} C_VEL
LIN {X 0,Y 361.862,Z 336.409,A -85,B 0,C 180,E1 -13177.222,E2 -13177.222} C_VEL
LIN {X 0,Y 361.834,Z 336.416,A -85,B 0,C 180,E1 -13180.755,E2 -13180.755} C_VEL
LIN {X 0,Y 361.843,Z 336.412,A -85,B 0,C 180,E1 -13184.364,E2 -13184.364} C_VEL
LIN {X 0,Y 361.834,Z 336.411,A -85,B 0,C 180,E1 -13187.568,E2 -13187.568} C_VEL
LIN {X 0,Y 361.869,Z 336.409,A -85,B 0,C 180,E1 -13190.973,E2 -13190.973} C_VEL
LIN {X 0,Y 361.872,Z 336.411,A -85,B 0,C 180,E1 -13194.655,E2 -13194.655} C_VEL
LIN {X 0,Y 361.835,Z 336.414,A -85,B 0,C 180,E1 -13198.37,E2 -13198.37} C_VEL
LIN {X 0,Y 361.906,Z 336.404,A -85,B 0,C 180,E1 -13202.221,E2 -13202.221} C_VEL
LIN {X 0,Y 361.926,Z 336.403,A -85,B 0,C 180,E1 -13204.71,E2 -13204.71} C_VEL
LIN {X 0,Y 361.89,Z 336.408,A -85,B 0,C 180,E1 -13208.347,E2 -13208.347} C_VEL
LIN {X 0,Y 361.964,Z 336.396,A -85,B 0,C 180,E1 -13212.061,E2 -13212.061} C_VEL
LIN {X 0,Y 361.995,Z 336.393,A -85,B 0,C 180,E1 -13216.101,E2 -13216.101} C_VEL
LIN {X 0,Y 362.03,Z 336.388,A -85,B 0,C 180,E1 -13219.938,E2 -13219.938} C_VEL
LIN {X 0,Y 362.149,Z 336.375,A -85,B 0,C 180,E1 -13222.193,E2 -13222.193} C_VEL
LIN {X 0,Y 362.116,Z 336.38,A -85,B 0,C 180,E1 -13224.431,E2 -13224.431} C_VEL
LIN {X 0,Y 362.28,Z 336.356,A -85,B 0,C 180,E1 -13227.777,E2 -13227.777} C_VEL
LIN {X 0,Y 362.425,Z 336.339,A -85,B 0,C 180,E1 -13230,E2 -13230} C_VEL
LIN {X 0,Y 362.28,Z 336.36,A -85,B 0,C 180,E1 -13232.224,E2 -13232.224} C_VEL
LIN {X 0,Y 362.17,Z 336.372,A -85,B 0,C 180,E1 -13236.686,E2 -13236.686} C_VEL
LIN {X 0,Y 362.072,Z 336.382,A -85,B 0,C 180,E1 -13238.934,E2 -13238.934} C_VEL
LIN {X 0,Y 361.958,Z 336.4,A -85,B 0,C 180,E1 -13242.333,E2 -13242.333} C_VEL
LIN {X 0,Y 361.96,Z 336.398,A -85,B 0,C 180,E1 -13244.621,E2 -13244.621} C_VEL
LIN {X 0,Y 361.957,Z 336.4,A -85,B 0,C 180,E1 -13248.1,E2 -13248.1} C_VEL
LIN {X 0,Y 361.89,Z 336.405,A -85,B 0,C 180,E1 -13251.653,E2 -13251.653} C_VEL
LIN {X 0,Y 361.927,Z 336.399,A -85,B 0,C 180,E1 -13255.291,E2 -13255.291} C_VEL
LIN {X 0,Y 361.907,Z 336.404,A -85,B 0,C 180,E1 -13257.78,E2 -13257.78} C_VEL
LIN {X 0,Y 361.836,Z 336.412,A -85,B 0,C 180,E1 -13261.63,E2 -13261.63} C_VEL
LIN {X 0,Y 361.874,Z 336.406,A -85,B 0,C 180,E1 -13265.346,E2 -13265.346} C_VEL
LIN {X 0,Y 361.847,Z 336.408,A -85,B 0,C 180,E1 -13267.765,E2 -13267.765} C_VEL
LIN {X 0,Y 361.183,Z 336.494,A -85,B 0,C 180,E1 -13268.694,E2 -13268.694} C_VEL
LIN {X 0,Y 358.325,Z 336.853,A -85,B 0,C 180,E1 -13270.205,E2 -13270.205} C_VEL
LIN {X 0,Y 355.904,Z 337.154,A -85,B 0,C 180,E1 -13271.428,E2 -13271.428} C_VEL
LIN {X 0,Y 354.868,Z 337.281,A -85,B 0,C 180,E1 -13272.374,E2 -13272.374} C_VEL
LIN {X 0,Y 354.786,Z 337.289,A -85,B 0,C 180,E1 -13272.695,E2 -13272.695} C_VEL
LIN {X 0,Y 354.767,Z 337.295,A -85,B 0,C 180,E1 -13276.104,E2 -13276.104} C_VEL
LIN {X 0,Y 354.788,Z 337.289,A -85,B 0,C 180,E1 -13279.18,E2 -13279.18} C_VEL
LIN {X 0,Y 354.807,Z 337.288,A -85,B 0,C 180,E1 -13282.403,E2 -13282.403} C_VEL
LIN {X 0,Y 354.812,Z 337.285,A -85,B 0,C 180,E1 -13284.942,E2 -13284.942} C_VEL
LIN {X 0,Y 354.794,Z 337.289,A -85,B 0,C 180,E1 -13288.406,E2 -13288.406} C_VEL
LIN {X 0,Y 354.927,Z 337.273,A -85,B 0,C 180,E1 -13291.406,E2 -13291.406} C_VEL
LIN {X 0,Y 360.978,Z 355.673,A -85,B 0,C 180,E1 -13292.167,E2 -13292.167} C_VEL
LIN {X 0,Y 359.534,Z 424.445,A -85,B 0,C 180,E1 -13293.909,E2 -13293.909} C_VEL
LIN {X 0,Y 359.341,Z 437.254,A -85,B 0,C 180,E1 -13294.449,E2 -13294.449} C_VEL
LIN {X 0,Y 358.881,Z 450.699,A -85,B 0,C 180,E1 -13295.255,E2 -13295.255} C_VEL
LIN {X 0,Y 358.353,Z 461.984,A -85,B 0,C 180,E1 -13296.141,E2 -13296.141} C_VEL
LIN {X 0,Y 357.745,Z 473.05,A -85,B 0,C 180,E1 -13297.24,E2 -13297.24} C_VEL
LIN {X 0,Y 357.06,Z 484.445,A -85,B 0,C 180,E1 -13298.646,E2 -13298.646} C_VEL
LIN {X 0,Y 356.33,Z 493.98,A -85,B 0,C 180,E1 -13300.11,E2 -13300.11} C_VEL
LIN {X 0,Y 355.784,Z 501.836,A -85,B 0,C 180,E1 -13301.576,E2 -13301.576} C_VEL
LIN {X 0,Y 355.276,Z 509.51,A -85,B 0,C 180,E1 -13303.332,E2 -13303.332} C_VEL
LIN {X 0,Y 354.909,Z 515.553,A -85,B 0,C 180,E1 -13305.083,E2 -13305.083} C_VEL
LIN {X 0,Y 354.682,Z 520.277,A -85,B 0,C 180,E1 -13306.829,E2 -13306.829} C_VEL
LIN {X 0,Y 354.479,Z 523.828,A -85,B 0,C 180,E1 -13308.565,E2 -13308.565} C_VEL
LIN {X 0,Y 354.454,Z 525.615,A -85,B 0,C 180,E1 -13309.721,E2 -13309.721} C_VEL
LIN {X 0,Y 354.503,Z 526.891,A -85,B 0,C 180,E1 -13310.875,E2 -13310.875} C_VEL
LIN {X 0,Y 354.638,Z 527.893,A -85,B 0,C 180,E1 -13312.255,E2 -13312.255} C_VEL
LIN {X 0,Y 354.812,Z 528.173,A -85,B 0,C 180,E1 -13314.317,E2 -13314.317} C_VEL
LIN {X 0,Y 354.878,Z 527.752,A -85,B 0,C 180,E1 -13315.457,E2 -13315.457} C_VEL
LIN {X 0,Y 355.201,Z 526.886,A -85,B 0,C 180,E1 -13316.598,E2 -13316.598} C_VEL
LIN {X 0,Y 355.519,Z 525.558,A -85,B 0,C 180,E1 -13317.735,E2 -13317.735} C_VEL
LIN {X 0,Y 356.118,Z 522.754,A -85,B 0,C 180,E1 -13319.435,E2 -13319.435} C_VEL
LIN {X 0,Y 356.837,Z 518.874,A -85,B 0,C 180,E1 -13321.129,E2 -13321.129} C_VEL
LIN {X 0,Y 357.747,Z 513.793,A -85,B 0,C 180,E1 -13322.816,E2 -13322.816} C_VEL
LIN {X 0,Y 358.769,Z 507.386,A -85,B 0,C 180,E1 -13324.495,E2 -13324.495} C_VEL
LIN {X 0,Y 360.006,Z 499.288,A -85,B 0,C 180,E1 -13326.164,E2 -13326.164} C_VEL
LIN {X 0,Y 361.047,Z 491.116,A -85,B 0,C 180,E1 -13327.551,E2 -13327.551} C_VEL
LIN {X 0,Y 362.34,Z 481.022,A -85,B 0,C 180,E1 -13328.927,E2 -13328.927} C_VEL
LIN {X 0,Y 363.44,Z 469.696,A -85,B 0,C 180,E1 -13330.164,E2 -13330.164} C_VEL
LIN {X 0,Y 364.422,Z 458.535,A -85,B 0,C 180,E1 -13331.12,E2 -13331.12} C_VEL
LIN {X 0,Y 365.168,Z 444.944,A -85,B 0,C 180,E1 -13332.011,E2 -13332.011} C_VEL
LIN {X 0,Y 365.618,Z 431.683,A -85,B 0,C 180,E1 -13332.63,E2 -13332.63} C_VEL
LIN {X 0,Y 366.361,Z 406.661,A -85,B 0,C 180,E1 -13333.384,E2 -13333.384} C_VEL
LIN {X 0,Y 368.488,Z 363.325,A -85,B 0,C 180,E1 -13334.609,E2 -13334.609} C_VEL
LIN {X 0,Y 364.15,Z 354.27,A -85,B 0,C 180,E1 -13335.41,E2 -13335.41} C_VEL
LIN {X 0,Y 358.939,Z 344.913,A -85,B 0,C 180,E1 -13336.378,E2 -13336.378} C_VEL
LIN {X 0,Y 356.703,Z 341.208,A -85,B 0,C 180,E1 -13336.814,E2 -13336.814} C_VEL
LIN {X 0,Y 355.234,Z 338.768,A -85,B 0,C 180,E1 -13337.11,E2 -13337.11} C_VEL
LIN {X 0,Y 354.858,Z 337.287,A -85,B 0,C 180,E1 -13337.238,E2 -13337.238} C_VEL
LIN {X 0,Y 354.82,Z 337.292,A -85,B 0,C 180,E1 -13341.417,E2 -13341.417} C_VEL
LIN {X 0,Y 354.809,Z 337.292,A -85,B 0,C 180,E1 -13344.581,E2 -13344.581} C_VEL
LIN {X 0,Y 354.8,Z 337.292,A -85,B 0,C 180,E1 -13348.386,E2 -13348.386} C_VEL
LIN {X 0,Y 354.79,Z 337.291,A -85,B 0,C 180,E1 -13352.334,E2 -13352.334} C_VEL
LIN {X 0,Y 354.822,Z 337.284,A -85,B 0,C 180,E1 -13355.698,E2 -13355.698} C_VEL
LIN {X 0,Y 354.772,Z 337.289,A -85,B 0,C 180,E1 -13359.413,E2 -13359.413} C_VEL
LIN {X 0,Y 354.786,Z 337.287,A -85,B 0,C 180,E1 -13362.866,E2 -13362.866} C_VEL
LIN {X 0,Y 354.769,Z 337.294,A -85,B 0,C 180,E1 -13366.103,E2 -13366.103} C_VEL
LIN {X 0,Y 354.769,Z 337.293,A -85,B 0,C 180,E1 -13369.176,E2 -13369.176} C_VEL
LIN {X 0,Y 354.804,Z 337.29,A -85,B 0,C 180,E1 -13372.404,E2 -13372.404} C_VEL
LIN {X 0,Y 354.922,Z 337.389,A -85,B 0,C 180,E1 -13376.306,E2 -13376.306} C_VEL
LIN {X 0,Y 358.784,Z 355.508,A -85,B 0,C 180,E1 -13380.068,E2 -13380.068} C_VEL
LIN {X 0,Y 359.892,Z 361.394,A -85,B 0,C 180,E1 -13381.247,E2 -13381.247} C_VEL
LIN {X 0,Y 358.362,Z 378.572,A -85,B 0,C 180,E1 -13384.44,E2 -13384.44} C_VEL
LIN {X 0,Y 358.126,Z 380.916,A -85,B 0,C 180,E1 -13384.869,E2 -13384.869} C_VEL
LIN {X 0,Y 361.879,Z 407.185,A -85,B 0,C 180,E1 -13386.236,E2 -13386.236} C_VEL
LIN {X 0,Y 364.174,Z 428.297,A -85,B 0,C 180,E1 -13387.185,E2 -13387.185} C_VEL
LIN {X 0,Y 365.362,Z 448.402,A -85,B 0,C 180,E1 -13387.966,E2 -13387.966} C_VEL
LIN {X 0,Y 363.046,Z 506.472,A -85,B 0,C 180,E1 -13389.607,E2 -13389.607} C_VEL
LIN {X 0,Y 361.952,Z 520.367,A -85,B 0,C 180,E1 -13390.209,E2 -13390.209} C_VEL
LIN {X 0,Y 360.477,Z 534.508,A -85,B 0,C 180,E1 -13391.087,E2 -13391.087} C_VEL
LIN {X 0,Y 359.132,Z 546.284,A -85,B 0,C 180,E1 -13392.048,E2 -13392.048} C_VEL
LIN {X 0,Y 357.698,Z 558.33,A -85,B 0,C 180,E1 -13393.3,E2 -13393.3} C_VEL
LIN {X 0,Y 356.406,Z 568.189,A -85,B 0,C 180,E1 -13394.561,E2 -13394.561} C_VEL
LIN {X 0,Y 355.459,Z 577.413,A -85,B 0,C 180,E1 -13396.013,E2 -13396.013} C_VEL
LIN {X 0,Y 354.586,Z 586.181,A -85,B 0,C 180,E1 -13397.698,E2 -13397.698} C_VEL
LIN {X 0,Y 354.027,Z 593.489,A -85,B 0,C 180,E1 -13399.419,E2 -13399.419} C_VEL
LIN {X 0,Y 353.826,Z 598.454,A -85,B 0,C 180,E1 -13400.857,E2 -13400.857} C_VEL
LIN {X 0,Y 353.754,Z 603.276,A -85,B 0,C 180,E1 -13402.58,E2 -13402.58} C_VEL
LIN {X 0,Y 353.905,Z 606.956,A -85,B 0,C 180,E1 -13404.301,E2 -13404.301} C_VEL
LIN {X 0,Y 354.043,Z 608.829,A -85,B 0,C 180,E1 -13405.446,E2 -13405.446} C_VEL
LIN {X 0,Y 354.157,Z 611.585,A -85,B 0,C 180,E1 -13407.725,E2 -13407.725} C_VEL
LIN {X 0,Y 354.174,Z 612.551,A -85,B 0,C 180,E1 -13408.863,E2 -13408.863} C_VEL
LIN {X 0,Y 354.209,Z 613.059,A -85,B 0,C 180,E1 -13410,E2 -13410} C_VEL
LIN {X 0,Y 354.104,Z 613.107,A -85,B 0,C 180,E1 -13411.137,E2 -13411.137} C_VEL
LIN {X 0,Y 354.051,Z 612.693,A -85,B 0,C 180,E1 -13412.275,E2 -13412.275} C_VEL
LIN {X 0,Y 354.071,Z 611.81,A -85,B 0,C 180,E1 -13413.414,E2 -13413.414} C_VEL
LIN {X 0,Y 353.903,Z 610.465,A -85,B 0,C 180,E1 -13414.556,E2 -13414.556} C_VEL
LIN {X 0,Y 353.729,Z 606.999,A -85,B 0,C 180,E1 -13416.574,E2 -13416.574} C_VEL
LIN {X 0,Y 353.704,Z 602.068,A -85,B 0,C 180,E1 -13418.57,E2 -13418.57} C_VEL
LIN {X 0,Y 353.947,Z 595.515,A -85,B 0,C 180,E1 -13420.583,E2 -13420.583} C_VEL
LIN {X 0,Y 354.591,Z 588.464,A -85,B 0,C 180,E1 -13422.302,E2 -13422.302} C_VEL
LIN {X 0,Y 355.53,Z 579.807,A -85,B 0,C 180,E1 -13424.009,E2 -13424.009} C_VEL
LIN {X 0,Y 356.509,Z 571.049,A -85,B 0,C 180,E1 -13425.434,E2 -13425.434} C_VEL
LIN {X 0,Y 357.891,Z 560.589,A -85,B 0,C 180,E1 -13426.837,E2 -13426.837} C_VEL
LIN {X 0,Y 359.502,Z 549.075,A -85,B 0,C 180,E1 -13428.08,E2 -13428.08} C_VEL
LIN {X 0,Y 361.035,Z 536.372,A -85,B 0,C 180,E1 -13429.177,E2 -13429.177} C_VEL
LIN {X 0,Y 362.613,Z 523.138,A -85,B 0,C 180,E1 -13430.048,E2 -13430.048} C_VEL
LIN {X 0,Y 363.856,Z 508.722,A -85,B 0,C 180,E1 -13430.751,E2 -13430.751} C_VEL
LIN {X 0,Y 364.754,Z 493.419,A -85,B 0,C 180,E1 -13431.252,E2 -13431.252} C_VEL
LIN {X 0,Y 366.883,Z 445.763,A -85,B 0,C 180,E1 -13432.651,E2 -13432.651} C_VEL
LIN {X 0,Y 365.755,Z 427.112,A -85,B 0,C 180,E1 -13433.433,E2 -13433.433} C_VEL
LIN {X 0,Y 364.192,Z 413.089,A -85,B 0,C 180,E1 -13434.126,E2 -13434.126} C_VEL
LIN {X 0,Y 361.077,Z 394.708,A -85,B 0,C 180,E1 -13435.214,E2 -13435.214} C_VEL
LIN {X 0,Y 359.783,Z 387.82,A -85,B 0,C 180,E1 -13435.686,E2 -13435.686} C_VEL
LIN {X 0,Y 362.409,Z 371.109,A -85,B 0,C 180,E1 -13439.23,E2 -13439.23} C_VEL
LIN {X 0,Y 362.767,Z 368.038,A -85,B 0,C 180,E1 -13439.924,E2 -13439.924} C_VEL
LIN {X 0,Y 361.382,Z 360.49,A -85,B 0,C 180,E1 -13441.992,E2 -13441.992} C_VEL
LIN {X 0,Y 359.277,Z 351.685,A -85,B 0,C 180,E1 -13444.756,E2 -13444.756} C_VEL
LIN {X 0,Y 357.574,Z 346.042,A -85,B 0,C 180,E1 -13446.831,E2 -13446.831} C_VEL
LIN {X 0,Y 355.539,Z 339.732,A -85,B 0,C 180,E1 -13449.563,E2 -13449.563} C_VEL
LIN {X 0,Y 354.767,Z 337.296,A -85,B 0,C 180,E1 -13450.824,E2 -13450.824} C_VEL
LIN {X 0,Y 354.768,Z 337.295,A -85,B 0,C 180,E1 -13453.896,E2 -13453.896} C_VEL
LIN {X 0,Y 354.79,Z 337.293,A -85,B 0,C 180,E1 -13457.661,E2 -13457.661} C_VEL
LIN {X 0,Y 354.787,Z 337.29,A -85,B 0,C 180,E1 -13460.662,E2 -13460.662} C_VEL
LIN {X 0,Y 354.82,Z 337.286,A -85,B 0,C 180,E1 -13464.301,E2 -13464.301} C_VEL
LIN {X 0,Y 354.788,Z 337.293,A -85,B 0,C 180,E1 -13467.666,E2 -13467.666} C_VEL
LIN {X 0,Y 354.798,Z 337.291,A -85,B 0,C 180,E1 -13471.614,E2 -13471.614} C_VEL
LIN {X 0,Y 354.805,Z 337.293,A -85,B 0,C 180,E1 -13475.419,E2 -13475.419} C_VEL
LIN {X 0,Y 354.84,Z 337.435,A -85,B 0,C 180,E1 -13475.906,E2 -13475.906} C_VEL
LIN {X 0,Y 355.796,Z 340.076,A -85,B 0,C 180,E1 -13476.186,E2 -13476.186} C_VEL
LIN {X 0,Y 357.562,Z 342.311,A -85,B 0,C 180,E1 -13476.562,E2 -13476.562} C_VEL
LIN {X 0,Y 359.611,Z 345.749,A -85,B 0,C 180,E1 -13477.025,E2 -13477.025} C_VEL
LIN {X 0,Y 366.045,Z 357.045,A -85,B 0,C 180,E1 -13478.377,E2 -13478.377} C_VEL
LIN {X 0,Y 369.847,Z 364.931,A -85,B 0,C 180,E1 -13479.153,E2 -13479.153} C_VEL
LIN {X 0,Y 366.635,Z 423.253,A -85,B 0,C 180,E1 -13480.925,E2 -13480.925} C_VEL
LIN {X 0,Y 366.281,Z 437.819,A -85,B 0,C 180,E1 -13481.47,E2 -13481.47} C_VEL
LIN {X 0,Y 365.664,Z 450.488,A -85,B 0,C 180,E1 -13482.162,E2 -13482.162} C_VEL
LIN {X 0,Y 364.793,Z 462.867,A -85,B 0,C 180,E1 -13483.058,E2 -13483.058} C_VEL
LIN {X 0,Y 363.656,Z 474.557,A -85,B 0,C 180,E1 -13484.158,E2 -13484.158} C_VEL
LIN {X 0,Y 362.514,Z 485.109,A -85,B 0,C 180,E1 -13485.402,E2 -13485.402} C_VEL
LIN {X 0,Y 361.253,Z 494.301,A -85,B 0,C 180,E1 -13486.739,E2 -13486.739} C_VEL
LIN {X 0,Y 359.871,Z 503.742,A -85,B 0,C 180,E1 -13488.452,E2 -13488.452} C_VEL
LIN {X 0,Y 358.644,Z 511.045,A -85,B 0,C 180,E1 -13490.126,E2 -13490.126} C_VEL
LIN {X 0,Y 357.464,Z 517.693,A -85,B 0,C 180,E1 -13492.089,E2 -13492.089} C_VEL
LIN {X 0,Y 356.589,Z 522.044,A -85,B 0,C 180,E1 -13493.776,E2 -13493.776} C_VEL
LIN {X 0,Y 355.884,Z 525.262,A -85,B 0,C 180,E1 -13495.469,E2 -13495.469} C_VEL
LIN {X 0,Y 355.51,Z 526.818,A -85,B 0,C 180,E1 -13496.599,E2 -13496.599} C_VEL
LIN {X 0,Y 355.265,Z 527.917,A -85,B 0,C 180,E1 -13497.732,E2 -13497.732} C_VEL
LIN {X 0,Y 355.024,Z 528.613,A -85,B 0,C 180,E1 -13498.865,E2 -13498.865} C_VEL
LIN {X 0,Y 354.896,Z 528.869,A -85,B 0,C 180,E1 -13499.999,E2 -13499.999} C_VEL
LIN {X 0,Y 354.666,Z 528.691,A -85,B 0,C 180,E1 -13501.135,E2 -13501.135} C_VEL
LIN {X 0,Y 354.314,Z 528.124,A -85,B 0,C 180,E1 -13502.273,E2 -13502.273} C_VEL
LIN {X 0,Y 354.349,Z 527.101,A -85,B 0,C 180,E1 -13503.411,E2 -13503.411} C_VEL
LIN {X 0,Y 354.548,Z 525.593,A -85,B 0,C 180,E1 -13504.547,E2 -13504.547} C_VEL
LIN {X 0,Y 354.703,Z 522.539,A -85,B 0,C 180,E1 -13506.256,E2 -13506.256} C_VEL
LIN {X 0,Y 354.763,Z 518.406,A -85,B 0,C 180,E1 -13507.971,E2 -13507.971} C_VEL
LIN {X 0,Y 355.126,Z 512.058,A -85,B 0,C 180,E1 -13509.971,E2 -13509.971} C_VEL
LIN {X 0,Y 355.541,Z 505.053,A -85,B 0,C 180,E1 -13511.689,E2 -13511.689} C_VEL
LIN {X 0,Y 356.132,Z 496.34,A -85,B 0,C 180,E1 -13513.407,E2 -13513.407} C_VEL
LIN {X 0,Y 356.677,Z 486.917,A -85,B 0,C 180,E1 -13514.916,E2 -13514.916} C_VEL
LIN {X 0,Y 357.317,Z 476.425,A -85,B 0,C 180,E1 -13516.276,E2 -13516.276} C_VEL
LIN {X 0,Y 357.929,Z 465.561,A -85,B 0,C 180,E1 -13517.423,E2 -13517.423} C_VEL
LIN {X 0,Y 358.474,Z 453.597,A -85,B 0,C 180,E1 -13518.429,E2 -13518.429} C_VEL
LIN {X 0,Y 359.057,Z 440.197,A -85,B 0,C 180,E1 -13519.287,E2 -13519.287} C_VEL
LIN {X 0,Y 359.308,Z 426.765,A -85,B 0,C 180,E1 -13519.903,E2 -13519.903} C_VEL
LIN {X 0,Y 359.585,Z 407.059,A -85,B 0,C 180,E1 -13520.467,E2 -13520.467} C_VEL
LIN {X 0,Y 360.729,Z 355.448,A -85,B 0,C 180,E1 -13521.802,E2 -13521.802} C_VEL
LIN {X 0,Y 354.859,Z 337.283,A -85,B 0,C 180,E1 -13522.548,E2 -13522.548} C_VEL
LIN {X 0,Y 354.899,Z 337.274,A -85,B 0,C 180,E1 -13525.827,E2 -13525.827} C_VEL
LIN {X 0,Y 354.853,Z 337.28,A -85,B 0,C 180,E1 -13529.678,E2 -13529.678} C_VEL
LIN {X 0,Y 354.805,Z 337.286,A -85,B 0,C 180,E1 -13533.701,E2 -13533.701} C_VEL
LIN {X 0,Y 354.796,Z 337.29,A -85,B 0,C 180,E1 -13536.459,E2 -13536.459} C_VEL
LIN {X 0,Y 354.822,Z 337.285,A -85,B 0,C 180,E1 -13539.423,E2 -13539.423} C_VEL
LIN {X 0,Y 354.786,Z 337.293,A -85,B 0,C 180,E1 -13542.867,E2 -13542.867} C_VEL
LIN {X 0,Y 354.766,Z 337.292,A -85,B 0,C 180,E1 -13546.103,E2 -13546.103} C_VEL
LIN {X 0,Y 354.787,Z 337.29,A -85,B 0,C 180,E1 -13549.179,E2 -13549.179} C_VEL
LIN {X 0,Y 354.81,Z 337.289,A -85,B 0,C 180,E1 -13552.401,E2 -13552.401} C_VEL
LIN {X 0,Y 354.81,Z 337.289,A -85,B 0,C 180,E1 -13554.941,E2 -13554.941} C_VEL
LIN {X 0,Y 354.791,Z 337.292,A -85,B 0,C 180,E1 -13558.405,E2 -13558.405} C_VEL
LIN {X 0,Y 354.844,Z 337.281,A -85,B 0,C 180,E1 -13561.618,E2 -13561.618} C_VEL
LIN {X 0,Y 354.896,Z 337.277,A -85,B 0,C 180,E1 -13564.172,E2 -13564.172} C_VEL
LIN {X 0,Y 354.833,Z 337.283,A -85,B 0,C 180,E1 -13567.894,E2 -13567.894} C_VEL
LIN {X 0,Y 354.919,Z 337.273,A -85,B 0,C 180,E1 -13571.892,E2 -13571.892} C_VEL
LIN {X 0,Y 354.94,Z 337.271,A -85,B 0,C 180,E1 -13575.981,E2 -13575.981} C_VEL
LIN {X 0,Y 354.977,Z 337.265,A -85,B 0,C 180,E1 -13579.736,E2 -13579.736} C_VEL
LIN {X 0,Y 355.112,Z 337.25,A -85,B 0,C 180,E1 -13582.037,E2 -13582.037} C_VEL
LIN {X 0,Y 355.09,Z 337.256,A -85,B 0,C 180,E1 -13584.321,E2 -13584.321} C_VEL
LIN {X 0,Y 355.243,Z 337.232,A -85,B 0,C 180,E1 -13587.733,E2 -13587.733} C_VEL
LIN {X 0,Y 355.395,Z 337.215,A -85,B 0,C 180,E1 -13590,E2 -13590} C_VEL
LIN {X 0,Y 355.243,Z 337.237,A -85,B 0,C 180,E1 -13592.268,E2 -13592.268} C_VEL
LIN {X 0,Y 355.136,Z 337.247,A -85,B 0,C 180,E1 -13596.819,E2 -13596.819} C_VEL
LIN {X 0,Y 355.013,Z 337.261,A -85,B 0,C 180,E1 -13599.113,E2 -13599.113} C_VEL
